gfCNCPoint2[28765] = {X 324.3107, Y 48.3200, Z -3.8333, A 0.000, B 0.000, C 0.000 }
gfCNCPoint2[28766] = {X 325.5555, Y 48.4004, Z -3.8333, A 0.000, B 0.000, C 0.000 }
gfCNCPoint2[28767] = {X 326.7797, Y 48.6402, Z -3.8333, A 0.000, B 0.000, C 0.000 }
gfCNCPoint2[28768] = {X 325.5882, Y 48.0963, Z -3.8333, A 0.000, B 0.000, C 0.000 }
gfCNCPoint2[28769] = {X 324.4810, Y 47.3966, Z -3.8333, A 0.000, B 0.000, C 0.000 }
gfCNCPoint2[28770] = {X 323.4784, Y 46.5538, Z -3.8333, A 0.000, B 0.000, C 0.000 }
gfCNCPoint2[28771] = {X 322.8382, Y 45.9295, Z -3.8333, A 0.000, B 0.000, C 0.000 }
gfCNCPoint2[28772] = {X 322.2180, Y 45.2650, Z -3.8333, A 0.000, B 0.000, C 0.000 }
gfCNCPoint2[28773] = {X 321.6628, Y 44.5452, Z -3.8333, A 0.000, B 0.000, C 0.000 }
gfCNCPoint2[28774] = {X 323.6300, Y 43.1703, Z -3.8333, A 0.000, B 0.000, C 0.000 }
gfCNCPoint2[28775] = {X 323.0063, Y 42.0918, Z -3.8333, A 0.000, B 0.000, C 0.000 }
gfCNCPoint2[28776] = {X 322.5757, Y 40.9227, Z -3.8333, A 0.000, B 0.000, C 0.000 }
gfCNCPoint2[28777] = {X 322.3506, Y 39.6973, Z -3.8333, A 0.000, B 0.000, C 0.000 }
gfCNCPoint2[28778] = {X 322.3379, Y 38.4514, Z -3.8333, A 0.000, B 0.000, C 0.000 }
gfCNCPoint2[28779] = {X 322.5377, Y 37.2217, Z -3.8333, A 0.000, B 0.000, C 0.000 }
gfCNCPoint2[28780] = {X 322.9443, Y 36.0440, Z -3.8333, A 0.000, B 0.000, C 0.000 }
gfCNCPoint2[28781] = {X 323.5458, Y 34.9529, Z -3.8333, A 0.000, B 0.000, C 0.000 }
gfCNCPoint2[28782] = {X 327.7841, Y 28.6157, Z -3.8333, A 0.000, B 0.000, C 0.000 }
gfCNCPoint2[28783] = {X 328.5200, Y 27.6906, Z -3.8333, A 0.000, B 0.000, C 0.000 }
gfCNCPoint2[28784] = {X 329.3960, Y 26.8968, Z -3.8333, A 0.000, B 0.000, C 0.000 }
gfCNCPoint2[28785] = {X 330.3889, Y 26.2552, Z -3.8333, A 0.000, B 0.000, C 0.000 }
gfCNCPoint2[28786] = {X 331.5063, Y 25.7713, Z -3.8333, A 0.000, B 0.000, C 0.000 }
gfCNCPoint2[28787] = {X 332.6887, Y 25.4804, Z -3.8333, A 0.000, B 0.000, C 0.000 }
gfCNCPoint2[28788] = {X 333.9031, Y 25.3907, Z -3.8333, A 0.000, B 0.000, C 0.000 }
gfCNCPoint2[28789] = {X 335.1154, Y 25.5046, Z -3.8333, A 0.000, B 0.000, C 0.000 }
gfCNCPoint2[28790] = {X 336.2918, Y 25.8191, Z -3.8333, A 0.000, B 0.000, C 0.000 }
gfCNCPoint2[28791] = {X 337.3993, Y 26.3252, Z -3.8333, A 0.000, B 0.000, C 0.000 }
gfCNCPoint2[28792] = {X 338.1754, Y 26.8291, Z -3.8333, A 0.000, B 0.000, C 0.000 }
gfCNCPoint2[28793] = {X 338.8813, Y 27.4275, Z -3.8333, A 0.000, B 0.000, C 0.000 }
gfCNCPoint2[28794] = {X 339.5028, Y 28.0267, Z -3.8333, A 0.000, B 0.000, C 0.000 }
gfCNCPoint2[28795] = {X 340.3314, Y 28.9977, Z -3.8333, A 0.000, B 0.000, C 0.000 }
gfCNCPoint2[28796] = {X 340.9777, Y 30.0985, Z -3.8333, A 0.000, B 0.000, C 0.000 }
gfCNCPoint2[28797] = {X 341.4218, Y 31.2952, Z -3.8333, A 0.000, B 0.000, C 0.000 }
gfCNCPoint2[28798] = {X 341.6500, Y 32.5511, Z -3.8333, A 0.000, B 0.000, C 0.000 }
gfCNCPoint2[28799] = {X 341.8446, Y 32.7091, Z -3.8333, A 0.000, B 0.000, C 0.000 }
gfCNCPoint2[28800] = {X 342.0414, Y 32.8643, Z -3.8333, A 0.000, B 0.000, C 0.000 }
gfCNCPoint2[28801] = {X 342.9843, Y 33.4816, Z -3.8333, A 0.000, B 0.000, C 0.000 }
gfCNCPoint2[28802] = {X 344.0076, Y 33.9537, Z -3.8333, A 0.000, B 0.000, C 0.000 }
gfCNCPoint2[28803] = {X 345.0891, Y 34.2705, Z -3.8333, A 0.000, B 0.000, C 0.000 }
gfCNCPoint2[28804] = {X 346.2053, Y 34.4251, Z -3.8333, A 0.000, B 0.000, C 0.000 }
gfCNCPoint2[28805] = {X 347.3322, Y 34.4141, Z -3.8333, A 0.000, B 0.000, C 0.000 }
gfCNCPoint2[28806] = {X 348.3018, Y 34.2887, Z -3.8333, A 0.000, B 0.000, C 0.000 }
gfCNCPoint2[28807] = {X 349.2376, Y 34.0059, Z -3.8333, A 0.000, B 0.000, C 0.000 }
gfCNCPoint2[28808] = {X 350.1143, Y 33.5732, Z -3.8333, A 0.000, B 0.000, C 0.000 }
gfCNCPoint2[28809] = {X 350.9081, Y 33.0025, Z -3.8333, A 0.000, B 0.000, C 0.000 }
gfCNCPoint2[28810] = {X 351.7847, Y 32.1513, Z -3.8333, A 0.000, B 0.000, C 0.000 }
gfCNCPoint2[28811] = {X 352.5434, Y 31.1936, Z -3.8333, A 0.000, B 0.000, C 0.000 }
gfCNCPoint2[28812] = {X 353.1716, Y 30.1456, Z -3.8333, A 0.000, B 0.000, C 0.000 }
gfCNCPoint2[28813] = {X 353.6586, Y 29.0250, Z -3.8333, A 0.000, B 0.000, C 0.000 }
gfCNCPoint2[28814] = {X 353.9962, Y 27.8507, Z -3.8333, A 0.000, B 0.000, C 0.000 }
gfCNCPoint2[28815] = {X 354.2236, Y 26.4407, Z -3.8333, A 0.000, B 0.000, C 0.000 }
gfCNCPoint2[28816] = {X 354.3157, Y 25.0155, Z -3.8333, A 0.000, B 0.000, C 0.000 }
gfCNCPoint2[28817] = {X 354.2717, Y 23.5880, Z -3.8333, A 0.000, B 0.000, C 0.000 }
gfCNCPoint2[28818] = {X 354.0919, Y 22.1712, Z -3.8333, A 0.000, B 0.000, C 0.000 }
gfCNCPoint2[28819] = {X 353.8393, Y 21.0759, Z -3.8333, A 0.000, B 0.000, C 0.000 }
gfCNCPoint2[28820] = {X 353.4527, Y 20.0204, Z -3.8333, A 0.000, B 0.000, C 0.000 }
gfCNCPoint2[28821] = {X 352.9380, Y 19.0210, Z -3.8333, A 0.000, B 0.000, C 0.000 }
gfCNCPoint2[28822] = {X 352.3033, Y 18.0933, Z -3.8333, A 0.000, B 0.000, C 0.000 }
gfCNCPoint2[28823] = {X 351.5364, Y 17.2660, Z -3.8333, A 0.000, B 0.000, C 0.000 }
gfCNCPoint2[28824] = {X 350.6339, Y 16.5894, Z -3.8333, A 0.000, B 0.000, C 0.000 }
gfCNCPoint2[28825] = {X 349.6248, Y 16.0851, Z -3.8333, A 0.000, B 0.000, C 0.000 }
gfCNCPoint2[28826] = {X 348.5418, Y 15.7695, Z -3.8333, A 0.000, B 0.000, C 0.000 }
gfCNCPoint2[28827] = {X 347.1561, Y 15.5988, Z -3.8333, A 0.000, B 0.000, C 0.000 }
gfCNCPoint2[28828] = {X 345.7600, Y 15.6149, Z -3.8333, A 0.000, B 0.000, C 0.000 }
gfCNCPoint2[28829] = {X 344.3786, Y 15.8174, Z -3.8333, A 0.000, B 0.000, C 0.000 }
gfCNCPoint2[28830] = {X 343.0366, Y 16.2027, Z -3.8333, A 0.000, B 0.000, C 0.000 }
gfCNCPoint2[28831] = {X 341.7582, Y 16.7639, Z -3.8333, A 0.000, B 0.000, C 0.000 }
gfCNCPoint2[28832] = {X 341.4305, Y 17.8589, Z -3.8333, A 0.000, B 0.000, C 0.000 }
gfCNCPoint2[28833] = {X 340.9355, Y 18.8891, Z -3.8333, A 0.000, B 0.000, C 0.000 }
gfCNCPoint2[28834] = {X 340.2853, Y 19.8292, Z -3.8333, A 0.000, B 0.000, C 0.000 }
gfCNCPoint2[28835] = {X 345.8671, Y 24.3770, Z -3.8333, A 0.000, B 0.000, C 0.000 }
gfCNCPoint2[28836] = {X 346.4659, Y 25.2133, Z -3.8333, A 0.000, B 0.000, C 0.000 }
gfCNCPoint2[28837] = {X 347.0039, Y 26.0900, Z -3.8333, A 0.000, B 0.000, C 0.000 }
gfCNCPoint2[28838] = {X 347.1178, Y 24.7341, Z -3.8333, A 0.000, B 0.000, C 0.000 }
gfCNCPoint2[28839] = {X 346.9938, Y 23.3790, Z -3.8333, A 0.000, B 0.000, C 0.000 }
gfCNCPoint2[28840] = {X 346.9498, Y 23.1696, Z -3.8333, A 0.000, B 0.000, C 0.000 }
gfCNCPoint2[28841] = {X 346.8818, Y 22.9666, Z -3.8333, A 0.000, B 0.000, C 0.000 }
gfCNCPoint2[28842] = {X 346.3957, Y 23.6871, Z -3.8333, A 0.000, B 0.000, C 0.000 }
gfCNCPoint2[28843] = {X 345.8671, Y 24.3770, Z -3.8333, A 0.000, B 0.000, C 0.000 }
gfCNCPoint2[28844] = {X 344.0065, Y 22.8611, Z -3.8333, A 0.000, B 0.000, C 0.000 }
gfCNCPoint2[28845] = {X 343.3271, Y 23.6263, Z -3.8333, A 0.000, B 0.000, C 0.000 }
gfCNCPoint2[28846] = {X 342.5854, Y 24.3313, Z -3.8333, A 0.000, B 0.000, C 0.000 }
gfCNCPoint2[28847] = {X 342.8589, Y 24.5949, Z -3.8333, A 0.000, B 0.000, C 0.000 }
gfCNCPoint2[28848] = {X 343.9809, Y 25.8612, Z -3.8333, A 0.000, B 0.000, C 0.000 }
gfCNCPoint2[28849] = {X 344.9149, Y 27.2717, Z -3.8333, A 0.000, B 0.000, C 0.000 }
gfCNCPoint2[28850] = {X 345.4668, Y 28.3751, Z -3.8333, A 0.000, B 0.000, C 0.000 }
gfCNCPoint2[28851] = {X 345.9032, Y 29.5290, Z -3.8333, A 0.000, B 0.000, C 0.000 }
gfCNCPoint2[28852] = {X 346.4601, Y 29.6317, Z -3.8333, A 0.000, B 0.000, C 0.000 }
gfCNCPoint2[28853] = {X 347.0263, Y 29.6224, Z -3.8333, A 0.000, B 0.000, C 0.000 }
gfCNCPoint2[28854] = {X 347.4358, Y 29.5572, Z -3.8333, A 0.000, B 0.000, C 0.000 }
gfCNCPoint2[28855] = {X 347.7945, Y 29.3494, Z -3.8333, A 0.000, B 0.000, C 0.000 }
gfCNCPoint2[28856] = {X 348.4750, Y 28.6296, Z -3.8333, A 0.000, B 0.000, C 0.000 }
gfCNCPoint2[28857] = {X 348.9857, Y 27.7810, Z -3.8333, A 0.000, B 0.000, C 0.000 }
gfCNCPoint2[28858] = {X 349.3032, Y 26.8428, Z -3.8333, A 0.000, B 0.000, C 0.000 }
gfCNCPoint2[28859] = {X 349.3374, Y 26.6713, Z -3.8333, A 0.000, B 0.000, C 0.000 }
gfCNCPoint2[28860] = {X 349.3687, Y 26.4992, Z -3.8333, A 0.000, B 0.000, C 0.000 }
gfCNCPoint2[28861] = {X 349.5021, Y 25.3279, Z -3.8333, A 0.000, B 0.000, C 0.000 }
gfCNCPoint2[28862] = {X 349.4993, Y 24.1490, Z -3.8333, A 0.000, B 0.000, C 0.000 }
gfCNCPoint2[28863] = {X 349.3602, Y 22.9783, Z -3.8333, A 0.000, B 0.000, C 0.000 }
gfCNCPoint2[28864] = {X 349.1884, Y 22.2867, Z -3.8333, A 0.000, B 0.000, C 0.000 }
gfCNCPoint2[28865] = {X 348.9031, Y 21.6337, Z -3.8333, A 0.000, B 0.000, C 0.000 }
gfCNCPoint2[28866] = {X 348.5124, Y 21.0377, Z -3.8333, A 0.000, B 0.000, C 0.000 }
gfCNCPoint2[28867] = {X 348.1200, Y 20.6785, Z -3.8333, A 0.000, B 0.000, C 0.000 }
gfCNCPoint2[28868] = {X 347.6259, Y 20.4813, Z -3.8333, A 0.000, B 0.000, C 0.000 }
gfCNCPoint2[28869] = {X 346.5728, Y 20.3828, Z -3.8333, A 0.000, B 0.000, C 0.000 }
gfCNCPoint2[28870] = {X 345.5198, Y 20.4831, Z -3.8333, A 0.000, B 0.000, C 0.000 }
gfCNCPoint2[28871] = {X 344.8328, Y 21.7164, Z -3.8333, A 0.000, B 0.000, C 0.000 }
gfCNCPoint2[28872] = {X 344.0065, Y 22.8611, Z -3.8333, A 0.000, B 0.000, C 0.000 }
gfCNCPoint2[28873] = {X 342.1459, Y 21.3451, Z -3.8333, A 0.000, B 0.000, C 0.000 }
gfCNCPoint2[28874] = {X 341.6015, Y 21.9583, Z -3.8333, A 0.000, B 0.000, C 0.000 }
gfCNCPoint2[28875] = {X 341.0072, Y 22.5232, Z -3.8333, A 0.000, B 0.000, C 0.000 }
gfCNCPoint2[28876] = {X 340.7216, Y 22.7630, Z -3.8333, A 0.000, B 0.000, C 0.000 }
gfCNCPoint2[28877] = {X 340.4270, Y 22.9916, Z -3.8333, A 0.000, B 0.000, C 0.000 }
gfCNCPoint2[28878] = {X 339.6615, Y 23.5549, Z -3.8333, A 0.000, B 0.000, C 0.000 }
gfCNCPoint2[28879] = {X 339.1299, Y 23.9121, Z -3.8333, A 0.000, B 0.000, C 0.000 }
gfCNCPoint2[28880] = {X 338.5759, Y 24.2333, Z -3.8333, A 0.000, B 0.000, C 0.000 }
gfCNCPoint2[28881] = {X 339.6078, Y 24.9035, Z -3.8333, A 0.000, B 0.000, C 0.000 }
gfCNCPoint2[28882] = {X 340.5464, Y 25.6991, Z -3.8333, A 0.000, B 0.000, C 0.000 }
gfCNCPoint2[28883] = {X 341.1848, Y 26.3148, Z -3.8333, A 0.000, B 0.000, C 0.000 }
gfCNCPoint2[28884] = {X 342.1201, Y 27.3790, Z -3.8333, A 0.000, B 0.000, C 0.000 }
gfCNCPoint2[28885] = {X 342.8900, Y 28.5683, Z -3.8333, A 0.000, B 0.000, C 0.000 }
gfCNCPoint2[28886] = {X 343.4780, Y 29.8572, Z -3.8333, A 0.000, B 0.000, C 0.000 }
gfCNCPoint2[28887] = {X 343.8716, Y 31.2182, Z -3.8333, A 0.000, B 0.000, C 0.000 }
gfCNCPoint2[28888] = {X 344.6368, Y 31.6212, Z -3.8333, A 0.000, B 0.000, C 0.000 }
gfCNCPoint2[28889] = {X 345.4577, Y 31.8932, Z -3.8333, A 0.000, B 0.000, C 0.000 }
gfCNCPoint2[28890] = {X 346.3121, Y 32.0269, Z -3.8333, A 0.000, B 0.000, C 0.000 }
gfCNCPoint2[28891] = {X 347.1768, Y 32.0187, Z -3.8333, A 0.000, B 0.000, C 0.000 }
gfCNCPoint2[28892] = {X 347.9590, Y 31.9040, Z -3.8333, A 0.000, B 0.000, C 0.000 }
gfCNCPoint2[28893] = {X 348.6962, Y 31.6182, Z -3.8333, A 0.000, B 0.000, C 0.000 }
gfCNCPoint2[28894] = {X 349.3514, Y 31.1758, Z -3.8333, A 0.000, B 0.000, C 0.000 }
gfCNCPoint2[28895] = {X 350.1528, Y 30.3722, Z -3.8333, A 0.000, B 0.000, C 0.000 }
gfCNCPoint2[28896] = {X 350.8138, Y 29.4496, Z -3.8333, A 0.000, B 0.000, C 0.000 }
gfCNCPoint2[28897] = {X 351.3172, Y 28.4324, Z -3.8333, A 0.000, B 0.000, C 0.000 }
gfCNCPoint2[28898] = {X 351.6496, Y 27.3472, Z -3.8333, A 0.000, B 0.000, C 0.000 }
gfCNCPoint2[28899] = {X 351.8779, Y 25.7641, Z -3.8333, A 0.000, B 0.000, C 0.000 }
gfCNCPoint2[28900] = {X 351.9036, Y 24.1648, Z -3.8333, A 0.000, B 0.000, C 0.000 }
gfCNCPoint2[28901] = {X 351.7261, Y 22.5752, Z -3.8333, A 0.000, B 0.000, C 0.000 }
gfCNCPoint2[28902] = {X 351.4573, Y 21.5045, Z -3.8333, A 0.000, B 0.000, C 0.000 }
gfCNCPoint2[28903] = {X 351.0147, Y 20.4931, Z -3.8333, A 0.000, B 0.000, C 0.000 }
gfCNCPoint2[28904] = {X 350.4107, Y 19.5691, Z -3.8333, A 0.000, B 0.000, C 0.000 }
gfCNCPoint2[28905] = {X 349.7597, Y 18.9043, Z -3.8333, A 0.000, B 0.000, C 0.000 }
gfCNCPoint2[28906] = {X 348.9692, Y 18.4138, Z -3.8333, A 0.000, B 0.000, C 0.000 }
gfCNCPoint2[28907] = {X 348.0845, Y 18.1256, Z -3.8333, A 0.000, B 0.000, C 0.000 }
gfCNCPoint2[28908] = {X 346.9930, Y 17.9935, Z -3.8333, A 0.000, B 0.000, C 0.000 }
gfCNCPoint2[28909] = {X 345.8937, Y 18.0119, Z -3.8333, A 0.000, B 0.000, C 0.000 }
gfCNCPoint2[28910] = {X 344.8073, Y 18.1805, Z -3.8333, A 0.000, B 0.000, C 0.000 }
gfCNCPoint2[28911] = {X 343.7541, Y 18.4960, Z -3.8333, A 0.000, B 0.000, C 0.000 }
gfCNCPoint2[28912] = {X 343.3269, Y 19.5045, Z -3.8333, A 0.000, B 0.000, C 0.000 }
gfCNCPoint2[28913] = {X 342.7886, Y 20.4583, Z -3.8333, A 0.000, B 0.000, C 0.000 }
gfCNCPoint2[28914] = {X 342.1459, Y 21.3451, Z -3.8333, A 0.000, B 0.000, C 0.000 }
gfCNCPoint2[28915] = {X 340.2853, Y 19.8292, Z -3.8333, A 0.000, B 0.000, C 0.000 }
gfCNCPoint2[28916] = {X 339.6794, Y 20.4860, Z -3.8333, A 0.000, B 0.000, C 0.000 }
gfCNCPoint2[28917] = {X 338.9976, Y 21.0636, Z -3.8333, A 0.000, B 0.000, C 0.000 }
gfCNCPoint2[28918] = {X 338.2497, Y 21.6140, Z -3.8333, A 0.000, B 0.000, C 0.000 }
gfCNCPoint2[28919] = {X 337.8538, Y 21.8795, Z -3.8333, A 0.000, B 0.000, C 0.000 }
gfCNCPoint2[28920] = {X 337.4413, Y 22.1185, Z -3.8333, A 0.000, B 0.000, C 0.000 }
gfCNCPoint2[28921] = {X 336.3239, Y 22.6023, Z -3.8333, A 0.000, B 0.000, C 0.000 }
gfCNCPoint2[28922] = {X 335.1415, Y 22.8932, Z -3.8333, A 0.000, B 0.000, C 0.000 }
gfCNCPoint2[28923] = {X 333.9271, Y 22.9829, Z -3.8333, A 0.000, B 0.000, C 0.000 }
gfCNCPoint2[28924] = {X 332.7148, Y 22.8690, Z -3.8333, A 0.000, B 0.000, C 0.000 }
gfCNCPoint2[28925] = {X 331.5384, Y 22.5546, Z -3.8333, A 0.000, B 0.000, C 0.000 }
gfCNCPoint2[28926] = {X 330.4309, Y 22.0485, Z -3.8333, A 0.000, B 0.000, C 0.000 }
gfCNCPoint2[28927] = {X 329.5143, Y 21.4374, Z -3.8333, A 0.000, B 0.000, C 0.000 }
gfCNCPoint2[28928] = {X 328.7005, Y 20.6949, Z -3.8333, A 0.000, B 0.000, C 0.000 }
gfCNCPoint2[28929] = {X 328.0080, Y 19.8382, Z -3.8333, A 0.000, B 0.000, C 0.000 }
gfCNCPoint2[28930] = {X 327.4528, Y 18.8869, Z -3.8333, A 0.000, B 0.000, C 0.000 }
gfCNCPoint2[28931] = {X 323.9321, Y 11.6443, Z -3.8333, A 0.000, B 0.000, C 0.000 }
gfCNCPoint2[28932] = {X 323.5337, Y 10.6422, Z -3.8333, A 0.000, B 0.000, C 0.000 }
gfCNCPoint2[28933] = {X 323.2878, Y 9.5922, Z -3.8333, A 0.000, B 0.000, C 0.000 }
gfCNCPoint2[28934] = {X 323.1997, Y 8.5174, Z -3.8333, A 0.000, B 0.000, C 0.000 }
gfCNCPoint2[28935] = {X 323.2713, Y 7.4413, Z -3.8333, A 0.000, B 0.000, C 0.000 }
gfCNCPoint2[28936] = {X 323.4720, Y 6.4885, Z -3.8333, A 0.000, B 0.000, C 0.000 }
gfCNCPoint2[28937] = {X 323.7980, Y 5.5709, Z -3.8333, A 0.000, B 0.000, C 0.000 }
gfCNCPoint2[28938] = {X 324.2435, Y 4.7050, Z -3.8333, A 0.000, B 0.000, C 0.000 }
gfCNCPoint2[28939] = {X 168.0205, Y 4.7050, Z -3.8333, A 0.000, B 0.000, C 0.000 }
gfCNCPoint2[28940] = {X 168.0205, Y 9.5050, Z -3.8333, A 0.000, B 0.000, C 0.000 }
gfCNCPoint2[28941] = {X 166.5360, Y 9.5050, Z -3.8333, A 0.000, B 0.000, C 0.000 }
gfCNCPoint2[28942] = {X 166.5855, Y 9.9931, Z -3.8333, A 0.000, B 0.000, C 0.000 }
gfCNCPoint2[28943] = {X 166.6021, Y 10.4835, Z -3.8333, A 0.000, B 0.000, C 0.000 }
gfCNCPoint2[28944] = {X 166.6021, Y 13.0969, Z -3.8333, A 0.000, B 0.000, C 0.000 }
gfCNCPoint2[28945] = {X 166.8569, Y 11.8210, Z -3.8333, A 0.000, B 0.000, C 0.000 }
gfCNCPoint2[28946] = {X 167.3348, Y 10.6108, Z -3.8333, A 0.000, B 0.000, C 0.000 }
gfCNCPoint2[28947] = {X 168.0205, Y 9.5050, Z -3.8333, A 0.000, B 0.000, C 0.000 }
gfCNCPoint2[28948] = {X 168.0205, Y 7.1050, Z -3.8333, A 0.000, B 0.000, C 0.000 }
gfCNCPoint2[28949] = {X 162.8435, Y 7.1050, Z -3.8333, A 0.000, B 0.000, C 0.000 }
gfCNCPoint2[28950] = {X 163.4703, Y 7.9131, Z -3.8333, A 0.000, B 0.000, C 0.000 }
gfCNCPoint2[28951] = {X 163.9149, Y 8.8341, Z -3.8333, A 0.000, B 0.000, C 0.000 }
gfCNCPoint2[28952] = {X 164.1578, Y 9.8276, Z -3.8333, A 0.000, B 0.000, C 0.000 }
gfCNCPoint2[28953] = {X 164.1910, Y 10.1548, Z -3.8333, A 0.000, B 0.000, C 0.000 }
gfCNCPoint2[28954] = {X 164.2021, Y 10.4835, Z -3.8333, A 0.000, B 0.000, C 0.000 }
gfCNCPoint2[28955] = {X 164.2021, Y 17.4615, Z -3.8333, A 0.000, B 0.000, C 0.000 }
gfCNCPoint2[28956] = {X 164.1139, Y 18.3848, Z -3.8333, A 0.000, B 0.000, C 0.000 }
gfCNCPoint2[28957] = {X 163.8527, Y 19.2747, Z -3.8333, A 0.000, B 0.000, C 0.000 }
gfCNCPoint2[28958] = {X 163.4279, Y 20.0992, Z -3.8333, A 0.000, B 0.000, C 0.000 }
gfCNCPoint2[28959] = {X 162.8547, Y 20.8283, Z -3.8333, A 0.000, B 0.000, C 0.000 }
gfCNCPoint2[28960] = {X 162.1539, Y 21.4359, Z -3.8333, A 0.000, B 0.000, C 0.000 }
gfCNCPoint2[28961] = {X 161.3508, Y 21.8998, Z -3.8333, A 0.000, B 0.000, C 0.000 }
gfCNCPoint2[28962] = {X 160.4745, Y 22.2035, Z -3.8333, A 0.000, B 0.000, C 0.000 }
gfCNCPoint2[28963] = {X 162.1747, Y 29.1999, Z -3.8333, A 0.000, B 0.000, C 0.000 }
gfCNCPoint2[28964] = {X 161.1123, Y 29.4081, Z -3.8333, A 0.000, B 0.000, C 0.000 }
gfCNCPoint2[28965] = {X 160.0356, Y 29.5204, Z -3.8333, A 0.000, B 0.000, C 0.000 }
gfCNCPoint2[28966] = {X 160.0350, Y 38.3365, Z -3.8333, A 0.000, B 0.000, C 0.000 }
gfCNCPoint2[28967] = {X 160.6830, Y 39.6933, Z -3.8333, A 0.000, B 0.000, C 0.000 }
gfCNCPoint2[28968] = {X 161.1580, Y 41.1200, Z -3.8333, A 0.000, B 0.000, C 0.000 }
gfCNCPoint2[28969] = {X 162.0480, Y 41.1200, Z -3.8333, A 0.000, B 0.000, C 0.000 }
gfCNCPoint2[28970] = {X 161.6737, Y 39.3706, Z -3.8333, A 0.000, B 0.000, C 0.000 }
gfCNCPoint2[28971] = {X 161.4498, Y 37.5957, Z -3.8333, A 0.000, B 0.000, C 0.000 }
gfCNCPoint2[28972] = {X 161.3316, Y 35.4804, Z -3.8333, A 0.000, B 0.000, C 0.000 }
gfCNCPoint2[28973] = {X 161.4138, Y 33.3634, Z -3.8333, A 0.000, B 0.000, C 0.000 }
gfCNCPoint2[28974] = {X 161.6957, Y 31.2636, Z -3.8333, A 0.000, B 0.000, C 0.000 }
gfCNCPoint2[28975] = {X 162.1747, Y 29.1999, Z -3.8333, A 0.000, B 0.000, C 0.000 }
gfCNCPoint2[28976] = {X 161.6080, Y 26.8678, Z -3.8333, A 0.000, B 0.000, C 0.000 }
gfCNCPoint2[28977] = {X 160.4732, Y 27.0728, Z -3.8333, A 0.000, B 0.000, C 0.000 }
gfCNCPoint2[28978] = {X 159.3221, Y 27.1415, Z -3.8333, A 0.000, B 0.000, C 0.000 }
gfCNCPoint2[28979] = {X 158.6554, Y 27.1415, Z -3.8333, A 0.000, B 0.000, C 0.000 }
gfCNCPoint2[28980] = {X 158.1448, Y 27.1258, Z -3.8333, A 0.000, B 0.000, C 0.000 }
gfCNCPoint2[28981] = {X 157.6357, Y 27.0833, Z -3.8333, A 0.000, B 0.000, C 0.000 }
gfCNCPoint2[28982] = {X 157.6349, Y 38.9960, Z -3.8333, A 0.000, B 0.000, C 0.000 }
gfCNCPoint2[28983] = {X 158.2188, Y 40.0484, Z -3.8333, A 0.000, B 0.000, C 0.000 }
gfCNCPoint2[28984] = {X 158.6680, Y 41.1649, Z -3.8333, A 0.000, B 0.000, C 0.000 }
gfCNCPoint2[28985] = {X 158.9759, Y 42.3283, Z -3.8333, A 0.000, B 0.000, C 0.000 }
gfCNCPoint2[28986] = {X 159.1375, Y 43.5209, Z -3.8333, A 0.000, B 0.000, C 0.000 }
gfCNCPoint2[28987] = {X 159.2980, Y 43.5200, Z -3.8333, A 0.000, B 0.000, C 0.000 }
gfCNCPoint2[28988] = {X 165.4299, Y 43.5200, Z -3.8333, A 0.000, B 0.000, C 0.000 }
gfCNCPoint2[28989] = {X 164.8363, Y 42.0419, Z -3.8333, A 0.000, B 0.000, C 0.000 }
gfCNCPoint2[28990] = {X 164.3714, Y 40.5184, Z -3.8333, A 0.000, B 0.000, C 0.000 }
gfCNCPoint2[28991] = {X 164.0379, Y 38.9571, Z -3.8333, A 0.000, B 0.000, C 0.000 }
gfCNCPoint2[28992] = {X 163.8396, Y 37.3729, Z -3.8333, A 0.000, B 0.000, C 0.000 }
gfCNCPoint2[28993] = {X 163.7317, Y 35.4783, Z -3.8333, A 0.000, B 0.000, C 0.000 }
gfCNCPoint2[28994] = {X 163.8039, Y 33.5820, Z -3.8333, A 0.000, B 0.000, C 0.000 }
gfCNCPoint2[28995] = {X 164.0555, Y 31.7011, Z -3.8333, A 0.000, B 0.000, C 0.000 }
gfCNCPoint2[28996] = {X 164.4843, Y 29.8525, Z -3.8333, A 0.000, B 0.000, C 0.000 }
gfCNCPoint2[28997] = {X 164.8363, Y 28.7332, Z -3.8333, A 0.000, B 0.000, C 0.000 }
gfCNCPoint2[28998] = {X 165.2534, Y 27.6365, Z -3.8333, A 0.000, B 0.000, C 0.000 }
gfCNCPoint2[28999] = {X 165.8700, Y 26.3057, Z -3.8333, A 0.000, B 0.000, C 0.000 }
gfCNCPoint2[29000] = {X 166.6043, Y 25.0361, Z -3.8333, A 0.000, B 0.000, C 0.000 }
gfCNCPoint2[29001] = {X 167.4503, Y 23.8379, Z -3.8333, A 0.000, B 0.000, C 0.000 }
gfCNCPoint2[29002] = {X 167.1640, Y 23.1367, Z -3.8333, A 0.000, B 0.000, C 0.000 }
gfCNCPoint2[29003] = {X 166.2873, Y 24.1837, Z -3.8333, A 0.000, B 0.000, C 0.000 }
gfCNCPoint2[29004] = {X 165.2721, Y 25.0970, Z -3.8333, A 0.000, B 0.000, C 0.000 }
gfCNCPoint2[29005] = {X 164.1384, Y 25.8583, Z -3.8333, A 0.000, B 0.000, C 0.000 }
gfCNCPoint2[29006] = {X 162.9089, Y 26.4525, Z -3.8333, A 0.000, B 0.000, C 0.000 }
gfCNCPoint2[29007] = {X 161.6080, Y 26.8678, Z -3.8333, A 0.000, B 0.000, C 0.000 }
gfCNCPoint2[29008] = {X 161.0412, Y 24.5356, Z -3.8333, A 0.000, B 0.000, C 0.000 }
gfCNCPoint2[29009] = {X 160.1878, Y 24.6899, Z -3.8333, A 0.000, B 0.000, C 0.000 }
gfCNCPoint2[29010] = {X 159.3221, Y 24.7415, Z -3.8333, A 0.000, B 0.000, C 0.000 }
gfCNCPoint2[29011] = {X 158.6660, Y 24.7415, Z -3.8333, A 0.000, B 0.000, C 0.000 }
gfCNCPoint2[29012] = {X 158.2815, Y 24.7297, Z -3.8333, A 0.000, B 0.000, C 0.000 }
gfCNCPoint2[29013] = {X 157.8982, Y 24.6977, Z -3.8333, A 0.000, B 0.000, C 0.000 }
gfCNCPoint2[29014] = {X 156.9779, Y 24.5364, Z -3.8333, A 0.000, B 0.000, C 0.000 }
gfCNCPoint2[29015] = {X 156.0856, Y 24.2591, Z -3.8333, A 0.000, B 0.000, C 0.000 }
gfCNCPoint2[29016] = {X 155.2360, Y 23.8704, Z -3.8333, A 0.000, B 0.000, C 0.000 }
gfCNCPoint2[29017] = {X 155.2349, Y 39.7518, Z -3.8333, A 0.000, B 0.000, C 0.000 }
gfCNCPoint2[29018] = {X 155.8256, Y 40.6437, Z -3.8333, A 0.000, B 0.000, C 0.000 }
gfCNCPoint2[29019] = {X 156.2800, Y 41.6123, Z -3.8333, A 0.000, B 0.000, C 0.000 }
gfCNCPoint2[29020] = {X 156.5883, Y 42.6368, Z -3.8333, A 0.000, B 0.000, C 0.000 }
gfCNCPoint2[29021] = {X 156.7438, Y 43.6953, Z -3.8333, A 0.000, B 0.000, C 0.000 }
gfCNCPoint2[29022] = {X 156.7578, Y 43.9475, Z -3.8333, A 0.000, B 0.000, C 0.000 }
gfCNCPoint2[29023] = {X 156.7631, Y 44.2001, Z -3.8333, A 0.000, B 0.000, C 0.000 }
gfCNCPoint2[29024] = {X 156.7629, Y 45.0587, Z -3.8333, A 0.000, B 0.000, C 0.000 }
gfCNCPoint2[29025] = {X 156.7352, Y 45.6370, Z -3.8333, A 0.000, B 0.000, C 0.000 }
gfCNCPoint2[29026] = {X 156.6616, Y 46.2112, Z -3.8333, A 0.000, B 0.000, C 0.000 }
gfCNCPoint2[29027] = {X 157.9053, Y 46.0006, Z -3.8333, A 0.000, B 0.000, C 0.000 }
gfCNCPoint2[29028] = {X 159.1641, Y 45.9207, Z -3.8333, A 0.000, B 0.000, C 0.000 }
gfCNCPoint2[29029] = {X 159.2310, Y 45.9202, Z -3.8333, A 0.000, B 0.000, C 0.000 }
gfCNCPoint2[29030] = {X 159.2980, Y 45.9200, Z -3.8333, A 0.000, B 0.000, C 0.000 }
gfCNCPoint2[29031] = {X 169.6833, Y 45.9200, Z -3.8333, A 0.000, B 0.000, C 0.000 }
gfCNCPoint2[29032] = {X 168.9026, Y 44.8481, Z -3.8333, A 0.000, B 0.000, C 0.000 }
gfCNCPoint2[29033] = {X 168.2121, Y 43.7159, Z -3.8333, A 0.000, B 0.000, C 0.000 }
gfCNCPoint2[29034] = {X 167.6167, Y 42.5310, Z -3.8333, A 0.000, B 0.000, C 0.000 }
gfCNCPoint2[29035] = {X 166.9487, Y 40.7946, Z -3.8333, A 0.000, B 0.000, C 0.000 }
gfCNCPoint2[29036] = {X 166.4842, Y 38.9930, Z -3.8333, A 0.000, B 0.000, C 0.000 }
gfCNCPoint2[29037] = {X 166.2294, Y 37.1501, Z -3.8333, A 0.000, B 0.000, C 0.000 }
gfCNCPoint2[29038] = {X 166.1311, Y 35.3976, Z -3.8333, A 0.000, B 0.000, C 0.000 }
gfCNCPoint2[29039] = {X 166.2079, Y 33.6441, Z -3.8333, A 0.000, B 0.000, C 0.000 }
gfCNCPoint2[29040] = {X 166.4591, Y 31.9069, Z -3.8333, A 0.000, B 0.000, C 0.000 }
gfCNCPoint2[29041] = {X 166.8820, Y 30.2034, Z -3.8333, A 0.000, B 0.000, C 0.000 }
gfCNCPoint2[29042] = {X 167.4726, Y 28.5505, Z -3.8333, A 0.000, B 0.000, C 0.000 }
gfCNCPoint2[29043] = {X 168.2334, Y 26.9813, Z -3.8333, A 0.000, B 0.000, C 0.000 }
gfCNCPoint2[29044] = {X 169.1857, Y 25.5205, Z -3.8333, A 0.000, B 0.000, C 0.000 }
gfCNCPoint2[29045] = {X 170.3144, Y 24.1911, Z -3.8333, A 0.000, B 0.000, C 0.000 }
gfCNCPoint2[29046] = {X 169.9865, Y 23.6224, Z -3.8333, A 0.000, B 0.000, C 0.000 }
gfCNCPoint2[29047] = {X 169.7113, Y 23.0264, Z -3.8333, A 0.000, B 0.000, C 0.000 }
gfCNCPoint2[29048] = {X 167.1001, Y 16.6309, Z -3.8333, A 0.000, B 0.000, C 0.000 }
gfCNCPoint2[29049] = {X 166.7820, Y 15.6636, Z -3.8333, A 0.000, B 0.000, C 0.000 }
gfCNCPoint2[29050] = {X 166.6021, Y 14.6613, Z -3.8333, A 0.000, B 0.000, C 0.000 }
gfCNCPoint2[29051] = {X 166.6021, Y 17.4615, Z -3.8333, A 0.000, B 0.000, C 0.000 }
gfCNCPoint2[29052] = {X 166.5130, Y 18.5970, Z -3.8333, A 0.000, B 0.000, C 0.000 }
gfCNCPoint2[29053] = {X 166.2479, Y 19.7047, Z -3.8333, A 0.000, B 0.000, C 0.000 }
gfCNCPoint2[29054] = {X 165.8132, Y 20.7575, Z -3.8333, A 0.000, B 0.000, C 0.000 }
gfCNCPoint2[29055] = {X 165.2197, Y 21.7296, Z -3.8333, A 0.000, B 0.000, C 0.000 }
gfCNCPoint2[29056] = {X 164.3787, Y 22.6988, Z -3.8333, A 0.000, B 0.000, C 0.000 }
gfCNCPoint2[29057] = {X 163.3807, Y 23.5052, Z -3.8333, A 0.000, B 0.000, C 0.000 }
gfCNCPoint2[29058] = {X 162.2565, Y 24.1239, Z -3.8333, A 0.000, B 0.000, C 0.000 }
gfCNCPoint2[29059] = {X 161.0412, Y 24.5356, Z -3.8333, A 0.000, B 0.000, C 0.000 }
gfCNCPoint2[29060] = {X 160.4745, Y 22.2035, Z -3.8333, A 0.000, B 0.000, C 0.000 }
gfCNCPoint2[29061] = {X 159.9024, Y 22.3069, Z -3.8333, A 0.000, B 0.000, C 0.000 }
gfCNCPoint2[29062] = {X 159.3221, Y 22.3415, Z -3.8333, A 0.000, B 0.000, C 0.000 }
gfCNCPoint2[29063] = {X 158.6766, Y 22.3415, Z -3.8333, A 0.000, B 0.000, C 0.000 }
gfCNCPoint2[29064] = {X 157.8799, Y 22.2730, Z -3.8333, A 0.000, B 0.000, C 0.000 }
gfCNCPoint2[29065] = {X 157.1047, Y 22.0761, Z -3.8333, A 0.000, B 0.000, C 0.000 }
gfCNCPoint2[29066] = {X 156.3718, Y 21.7562, Z -3.8333, A 0.000, B 0.000, C 0.000 }
gfCNCPoint2[29067] = {X 155.5229, Y 21.1783, Z -3.8333, A 0.000, B 0.000, C 0.000 }
gfCNCPoint2[29068] = {X 154.8126, Y 20.4367, Z -3.8333, A 0.000, B 0.000, C 0.000 }
gfCNCPoint2[29069] = {X 152.8362, Y 20.4376, Z -3.8333, A 0.000, B 0.000, C 0.000 }
gfCNCPoint2[29070] = {X 152.8348, Y 40.6542, Z -3.8333, A 0.000, B 0.000, C 0.000 }
gfCNCPoint2[29071] = {X 153.1753, Y 41.0225, Z -3.8333, A 0.000, B 0.000, C 0.000 }
gfCNCPoint2[29072] = {X 153.6797, Y 41.7264, Z -3.8333, A 0.000, B 0.000, C 0.000 }
gfCNCPoint2[29073] = {X 154.0528, Y 42.5079, Z -3.8333, A 0.000, B 0.000, C 0.000 }
gfCNCPoint2[29074] = {X 154.2830, Y 43.3428, Z -3.8333, A 0.000, B 0.000, C 0.000 }
gfCNCPoint2[29075] = {X 154.3631, Y 44.2051, Z -3.8333, A 0.000, B 0.000, C 0.000 }
gfCNCPoint2[29076] = {X 154.3629, Y 45.0469, Z -3.8333, A 0.000, B 0.000, C 0.000 }
gfCNCPoint2[29077] = {X 154.3441, Y 45.4307, Z -3.8333, A 0.000, B 0.000, C 0.000 }
gfCNCPoint2[29078] = {X 154.2951, Y 45.8119, Z -3.8333, A 0.000, B 0.000, C 0.000 }
gfCNCPoint2[29079] = {X 154.0370, Y 46.7541, Z -3.8333, A 0.000, B 0.000, C 0.000 }
gfCNCPoint2[29080] = {X 153.5963, Y 47.6260, Z -3.8333, A 0.000, B 0.000, C 0.000 }
gfCNCPoint2[29081] = {X 152.9909, Y 48.3926, Z -3.8333, A 0.000, B 0.000, C 0.000 }
gfCNCPoint2[29082] = {X 152.2448, Y 49.0233, Z -3.8333, A 0.000, B 0.000, C 0.000 }
gfCNCPoint2[29083] = {X 151.3881, Y 49.4928, Z -3.8333, A 0.000, B 0.000, C 0.000 }
gfCNCPoint2[29084] = {X 150.4551, Y 49.7822, Z -3.8333, A 0.000, B 0.000, C 0.000 }
gfCNCPoint2[29085] = {X 149.4831, Y 49.8800, Z -3.8333, A 0.000, B 0.000, C 0.000 }
gfCNCPoint2[29086] = {X 143.0396, Y 49.8800, Z -3.8333, A 0.000, B 0.000, C 0.000 }
gfCNCPoint2[29087] = {X 142.0923, Y 49.7872, Z -3.8333, A 0.000, B 0.000, C 0.000 }
gfCNCPoint2[29088] = {X 141.1811, Y 49.5122, Z -3.8333, A 0.000, B 0.000, C 0.000 }
gfCNCPoint2[29089] = {X 140.3405, Y 49.0656, Z -3.8333, A 0.000, B 0.000, C 0.000 }
gfCNCPoint2[29090] = {X 139.6026, Y 48.4643, Z -3.8333, A 0.000, B 0.000, C 0.000 }
gfCNCPoint2[29091] = {X 138.9955, Y 47.7312, Z -3.8333, A 0.000, B 0.000, C 0.000 }
gfCNCPoint2[29092] = {X 138.5423, Y 46.8942, Z -3.8333, A 0.000, B 0.000, C 0.000 }
gfCNCPoint2[29093] = {X 138.2601, Y 45.9852, Z -3.8333, A 0.000, B 0.000, C 0.000 }
gfCNCPoint2[29094] = {X 138.1598, Y 45.0386, Z -3.8333, A 0.000, B 0.000, C 0.000 }
gfCNCPoint2[29095] = {X 138.1601, Y 44.1416, Z -3.8333, A 0.000, B 0.000, C 0.000 }
gfCNCPoint2[29096] = {X 138.2148, Y 43.4769, Z -3.8333, A 0.000, B 0.000, C 0.000 }
gfCNCPoint2[29097] = {X 138.3597, Y 42.8258, Z -3.8333, A 0.000, B 0.000, C 0.000 }
gfCNCPoint2[29098] = {X 129.1532, Y 40.1052, Z -3.8333, A 0.000, B 0.000, C 0.000 }
gfCNCPoint2[29099] = {X 129.5665, Y 38.9035, Z -3.8333, A 0.000, B 0.000, C 0.000 }
gfCNCPoint2[29100] = {X 130.0836, Y 37.7426, Z -3.8333, A 0.000, B 0.000, C 0.000 }
gfCNCPoint2[29101] = {X 130.0836, Y 31.6021, Z -3.8333, A 0.000, B 0.000, C 0.000 }
gfCNCPoint2[29102] = {X 129.2061, Y 31.3797, Z -3.8333, A 0.000, B 0.000, C 0.000 }
gfCNCPoint2[29103] = {X 128.3442, Y 31.1029, Z -3.8333, A 0.000, B 0.000, C 0.000 }
gfCNCPoint2[29104] = {X 128.3439, Y 38.3287, Z -3.8333, A 0.000, B 0.000, C 0.000 }
gfCNCPoint2[29105] = {X 128.7845, Y 39.2006, Z -3.8333, A 0.000, B 0.000, C 0.000 }
gfCNCPoint2[29106] = {X 129.1532, Y 40.1052, Z -3.8333, A 0.000, B 0.000, C 0.000 }
gfCNCPoint2[29107] = {X 131.4548, Y 40.7854, Z -3.8333, A 0.000, B 0.000, C 0.000 }
gfCNCPoint2[29108] = {X 131.9017, Y 39.5320, Z -3.8333, A 0.000, B 0.000, C 0.000 }
gfCNCPoint2[29109] = {X 132.4836, Y 38.3354, Z -3.8333, A 0.000, B 0.000, C 0.000 }
gfCNCPoint2[29110] = {X 132.4836, Y 29.5202, Z -3.8333, A 0.000, B 0.000, C 0.000 }
gfCNCPoint2[29111] = {X 131.3524, Y 29.3993, Z -3.8333, A 0.000, B 0.000, C 0.000 }
gfCNCPoint2[29112] = {X 130.2377, Y 29.1725, Z -3.8333, A 0.000, B 0.000, C 0.000 }
gfCNCPoint2[29113] = {X 129.1492, Y 28.8419, Z -3.8333, A 0.000, B 0.000, C 0.000 }
gfCNCPoint2[29114] = {X 128.0248, Y 28.3765, Z -3.8333, A 0.000, B 0.000, C 0.000 }
gfCNCPoint2[29115] = {X 126.9529, Y 27.8004, Z -3.8333, A 0.000, B 0.000, C 0.000 }
gfCNCPoint2[29116] = {X 125.9444, Y 27.1194, Z -3.8333, A 0.000, B 0.000, C 0.000 }
gfCNCPoint2[29117] = {X 125.9438, Y 38.9893, Z -3.8333, A 0.000, B 0.000, C 0.000 }
gfCNCPoint2[29118] = {X 126.4738, Y 39.9284, Z -3.8333, A 0.000, B 0.000, C 0.000 }
gfCNCPoint2[29119] = {X 126.8960, Y 40.9205, Z -3.8333, A 0.000, B 0.000, C 0.000 }
gfCNCPoint2[29120] = {X 127.2098, Y 41.9730, Z -3.8333, A 0.000, B 0.000, C 0.000 }
gfCNCPoint2[29121] = {X 127.4025, Y 43.0542, Z -3.8333, A 0.000, B 0.000, C 0.000 }
gfCNCPoint2[29122] = {X 127.4714, Y 44.1502, Z -3.8333, A 0.000, B 0.000, C 0.000 }
gfCNCPoint2[29123] = {X 127.4716, Y 45.0000, Z -3.8333, A 0.000, B 0.000, C 0.000 }
gfCNCPoint2[29124] = {X 127.4070, Y 46.1159, Z -3.8333, A 0.000, B 0.000, C 0.000 }
gfCNCPoint2[29125] = {X 127.2143, Y 47.2168, Z -3.8333, A 0.000, B 0.000, C 0.000 }
gfCNCPoint2[29126] = {X 126.8960, Y 48.2883, Z -3.8333, A 0.000, B 0.000, C 0.000 }
gfCNCPoint2[29127] = {X 126.2883, Y 49.6376, Z -3.8333, A 0.000, B 0.000, C 0.000 }
gfCNCPoint2[29128] = {X 125.4821, Y 50.8786, Z -3.8333, A 0.000, B 0.000, C 0.000 }
gfCNCPoint2[29129] = {X 124.4962, Y 51.9821, Z -3.8333, A 0.000, B 0.000, C 0.000 }
gfCNCPoint2[29130] = {X 123.3536, Y 52.9225, Z -3.8333, A 0.000, B 0.000, C 0.000 }
gfCNCPoint2[29131] = {X 122.0810, Y 53.6778, Z -3.8333, A 0.000, B 0.000, C 0.000 }
gfCNCPoint2[29132] = {X 120.7081, Y 54.2302, Z -3.8333, A 0.000, B 0.000, C 0.000 }
gfCNCPoint2[29133] = {X 119.2671, Y 54.5669, Z -3.8333, A 0.000, B 0.000, C 0.000 }
gfCNCPoint2[29134] = {X 117.7916, Y 54.6800, Z -3.8333, A 0.000, B 0.000, C 0.000 }
gfCNCPoint2[29135] = {X 111.9185, Y 54.6800, Z -3.8333, A 0.000, B 0.000, C 0.000 }
gfCNCPoint2[29136] = {X 110.6386, Y 54.5950, Z -3.8333, A 0.000, B 0.000, C 0.000 }
gfCNCPoint2[29137] = {X 109.3812, Y 54.3415, Z -3.8333, A 0.000, B 0.000, C 0.000 }
gfCNCPoint2[29138] = {X 108.1683, Y 53.9240, Z -3.8333, A 0.000, B 0.000, C 0.000 }
gfCNCPoint2[29139] = {X 107.0213, Y 53.3498, Z -3.8333, A 0.000, B 0.000, C 0.000 }
gfCNCPoint2[29140] = {X 106.6480, Y 53.5578, Z -3.8333, A 0.000, B 0.000, C 0.000 }
gfCNCPoint2[29141] = {X 106.2658, Y 53.7492, Z -3.8333, A 0.000, B 0.000, C 0.000 }
gfCNCPoint2[29142] = {X 105.0149, Y 54.2383, Z -3.8333, A 0.000, B 0.000, C 0.000 }
gfCNCPoint2[29143] = {X 103.7084, Y 54.5495, Z -3.8333, A 0.000, B 0.000, C 0.000 }
gfCNCPoint2[29144] = {X 102.3713, Y 54.6768, Z -3.8333, A 0.000, B 0.000, C 0.000 }
gfCNCPoint2[29145] = {X 101.0295, Y 54.6179, Z -3.8333, A 0.000, B 0.000, C 0.000 }
gfCNCPoint2[29146] = {X 99.7088, Y 54.3738, Z -3.8333, A 0.000, B 0.000, C 0.000 }
gfCNCPoint2[29147] = {X 98.4345, Y 53.9493, Z -3.8333, A 0.000, B 0.000, C 0.000 }
gfCNCPoint2[29148] = {X 97.2313, Y 53.3524, Z -3.8333, A 0.000, B 0.000, C 0.000 }
gfCNCPoint2[29149] = {X 96.0852, Y 53.9255, Z -3.8333, A 0.000, B 0.000, C 0.000 }
gfCNCPoint2[29150] = {X 94.8734, Y 54.3422, Z -3.8333, A 0.000, B 0.000, C 0.000 }
gfCNCPoint2[29151] = {X 93.6172, Y 54.5952, Z -3.8333, A 0.000, B 0.000, C 0.000 }
gfCNCPoint2[29152] = {X 92.3385, Y 54.6800, Z -3.8333, A 0.000, B 0.000, C 0.000 }
gfCNCPoint2[29153] = {X 85.8951, Y 54.6800, Z -3.8333, A 0.000, B 0.000, C 0.000 }
gfCNCPoint2[29154] = {X 84.6159, Y 54.5951, Z -3.8333, A 0.000, B 0.000, C 0.000 }
gfCNCPoint2[29155] = {X 83.3592, Y 54.3419, Z -3.8333, A 0.000, B 0.000, C 0.000 }
gfCNCPoint2[29156] = {X 82.1469, Y 53.9249, Z -3.8333, A 0.000, B 0.000, C 0.000 }
gfCNCPoint2[29157] = {X 81.0644, Y 55.1572, Z -3.8333, A 0.000, B 0.000, C 0.000 }
gfCNCPoint2[29158] = {X 79.8495, Y 56.2591, Z -3.8333, A 0.000, B 0.000, C 0.000 }
gfCNCPoint2[29159] = {X 78.5178, Y 57.2166, Z -3.8333, A 0.000, B 0.000, C 0.000 }
gfCNCPoint2[29160] = {X 77.0863, Y 58.0174, Z -3.8333, A 0.000, B 0.000, C 0.000 }
gfCNCPoint2[29161] = {X 75.5734, Y 58.6511, Z -3.8333, A 0.000, B 0.000, C 0.000 }
gfCNCPoint2[29162] = {X 73.9986, Y 59.1096, Z -3.8333, A 0.000, B 0.000, C 0.000 }
gfCNCPoint2[29163] = {X 72.3820, Y 59.3871, Z -3.8333, A 0.000, B 0.000, C 0.000 }
gfCNCPoint2[29164] = {X 70.7445, Y 59.4800, Z -3.8333, A 0.000, B 0.000, C 0.000 }
gfCNCPoint2[29165] = {X 64.1851, Y 59.4800, Z -3.8333, A 0.000, B 0.000, C 0.000 }
gfCNCPoint2[29166] = {X 62.4203, Y 59.3720, Z -3.8333, A 0.000, B 0.000, C 0.000 }
gfCNCPoint2[29167] = {X 60.6818, Y 59.0498, Z -3.8333, A 0.000, B 0.000, C 0.000 }
gfCNCPoint2[29168] = {X 58.9955, Y 58.5181, Z -3.8333, A 0.000, B 0.000, C 0.000 }
gfCNCPoint2[29169] = {X 57.3866, Y 57.7848, Z -3.8333, A 0.000, B 0.000, C 0.000 }
gfCNCPoint2[29170] = {X 55.8790, Y 56.8608, Z -3.8333, A 0.000, B 0.000, C 0.000 }
gfCNCPoint2[29171] = {X 54.3715, Y 57.7848, Z -3.8333, A 0.000, B 0.000, C 0.000 }
gfCNCPoint2[29172] = {X 52.7626, Y 58.5181, Z -3.8333, A 0.000, B 0.000, C 0.000 }
gfCNCPoint2[29173] = {X 51.0763, Y 59.0498, Z -3.8333, A 0.000, B 0.000, C 0.000 }
gfCNCPoint2[29174] = {X 49.3378, Y 59.3720, Z -3.8333, A 0.000, B 0.000, C 0.000 }
gfCNCPoint2[29175] = {X 47.5729, Y 59.4800, Z -3.8333, A 0.000, B 0.000, C 0.000 }
gfCNCPoint2[29176] = {X 40.6393, Y 59.4800, Z -3.8333, A 0.000, B 0.000, C 0.000 }
gfCNCPoint2[29177] = {X 38.9796, Y 59.3846, Z -3.8333, A 0.000, B 0.000, C 0.000 }
gfCNCPoint2[29178] = {X 37.3418, Y 59.0995, Z -3.8333, A 0.000, B 0.000, C 0.000 }
gfCNCPoint2[29179] = {X 35.7474, Y 58.6286, Z -3.8333, A 0.000, B 0.000, C 0.000 }
gfCNCPoint2[29180] = {X 34.0329, Y 59.4869, Z -3.8333, A 0.000, B 0.000, C 0.000 }
gfCNCPoint2[29181] = {X 32.2400, Y 60.1662, Z -3.8333, A 0.000, B 0.000, C 0.000 }
gfCNCPoint2[29182] = {X 30.3872, Y 60.6596, Z -3.8333, A 0.000, B 0.000, C 0.000 }
gfCNCPoint2[29183] = {X 28.4938, Y 60.9618, Z -3.8333, A 0.000, B 0.000, C 0.000 }
gfCNCPoint2[29184] = {X 26.3374, Y 61.8556, Z -3.8333, A 0.000, B 0.000, C 0.000 }
gfCNCPoint2[29185] = {X 24.1361, Y 62.6325, Z -3.8333, A 0.000, B 0.000, C 0.000 }
gfCNCPoint2[29186] = {X 21.7294, Y 63.3344, Z -3.8333, A 0.000, B 0.000, C 0.000 }
gfCNCPoint2[29187] = {X 19.2810, Y 63.8733, Z -3.8333, A 0.000, B 0.000, C 0.000 }
gfCNCPoint2[29188] = {X 16.8020, Y 64.2465, Z -3.8333, A 0.000, B 0.000, C 0.000 }
gfCNCPoint2[29189] = {X 14.3035, Y 64.4526, Z -3.8333, A 0.000, B 0.000, C 0.000 }
gfCNCPoint2[29190] = {X 14.3035, Y 85.6950, Z -3.8333, A 0.000, B 0.000, C 0.000 }
gfCNCPoint2[29191] = {X 112.5232, Y 85.6950, Z -3.8333, A 0.000, B 0.000, C 0.000 }
gfCNCPoint2[29192] = {X 113.6258, Y 84.5917, Z -3.8333, A 0.000, B 0.000, C 0.000 }
gfCNCPoint2[29193] = {X 114.8256, Y 83.5948, Z -3.8333, A 0.000, B 0.000, C 0.000 }
gfCNCPoint2[29194] = {X 116.1122, Y 82.7130, Z -3.8333, A 0.000, B 0.000, C 0.000 }
gfCNCPoint2[29195] = {X 117.4748, Y 81.9537, Z -3.8333, A 0.000, B 0.000, C 0.000 }
gfCNCPoint2[29196] = {X 111.0539, Y 69.0645, Z -3.8333, A 0.000, B 0.000, C 0.000 }
gfCNCPoint2[29197] = {X 109.0273, Y 68.9058, Z -3.8333, A 0.000, B 0.000, C 0.000 }
gfCNCPoint2[29198] = {X 107.0213, Y 68.5768, Z -3.8333, A 0.000, B 0.000, C 0.000 }
gfCNCPoint2[29199] = {X 105.0765, Y 68.8983, Z -3.8333, A 0.000, B 0.000, C 0.000 }
gfCNCPoint2[29200] = {X 103.1119, Y 69.0597, Z -3.8333, A 0.000, B 0.000, C 0.000 }
gfCNCPoint2[29201] = {X 101.1407, Y 69.0599, Z -3.8333, A 0.000, B 0.000, C 0.000 }
gfCNCPoint2[29202] = {X 99.1761, Y 68.8989, Z -3.8333, A 0.000, B 0.000, C 0.000 }
gfCNCPoint2[29203] = {X 97.2313, Y 68.5777, Z -3.8333, A 0.000, B 0.000, C 0.000 }
gfCNCPoint2[29204] = {X 95.6131, Y 68.8563, Z -3.8333, A 0.000, B 0.000, C 0.000 }
gfCNCPoint2[29205] = {X 93.9796, Y 69.0240, Z -3.8333, A 0.000, B 0.000, C 0.000 }
gfCNCPoint2[29206] = {X 92.3385, Y 69.0800, Z -3.8333, A 0.000, B 0.000, C 0.000 }
gfCNCPoint2[29207] = {X 86.6884, Y 69.0800, Z -3.8333, A 0.000, B 0.000, C 0.000 }
gfCNCPoint2[29208] = {X 84.7317, Y 70.2668, Z -3.8333, A 0.000, B 0.000, C 0.000 }
gfCNCPoint2[29209] = {X 82.6871, Y 71.2950, Z -3.8333, A 0.000, B 0.000, C 0.000 }
gfCNCPoint2[29210] = {X 107.2684, Y 71.2950, Z -3.8333, A 0.000, B 0.000, C 0.000 }
gfCNCPoint2[29211] = {X 109.1219, Y 70.1132, Z -3.8333, A 0.000, B 0.000, C 0.000 }
gfCNCPoint2[29212] = {X 111.0539, Y 69.0645, Z -3.8333, A 0.000, B 0.000, C 0.000 }
gfCNCPoint2[29213] = {X 112.1240, Y 71.2127, Z -3.8333, A 0.000, B 0.000, C 0.000 }
gfCNCPoint2[29214] = {X 113.1266, Y 70.7371, Z -3.8333, A 0.000, B 0.000, C 0.000 }
gfCNCPoint2[29215] = {X 114.1466, Y 70.3003, Z -3.8333, A 0.000, B 0.000, C 0.000 }
gfCNCPoint2[29216] = {X 117.4434, Y 66.6800, Z -3.8333, A 0.000, B 0.000, C 0.000 }
gfCNCPoint2[29217] = {X 111.9185, Y 66.6800, Z -3.8333, A 0.000, B 0.000, C 0.000 }
gfCNCPoint2[29218] = {X 111.5292, Y 66.6765, Z -3.8333, A 0.000, B 0.000, C 0.000 }
gfCNCPoint2[29219] = {X 111.1400, Y 66.6660, Z -3.8333, A 0.000, B 0.000, C 0.000 }
gfCNCPoint2[29220] = {X 109.0675, Y 66.4917, Z -3.8333, A 0.000, B 0.000, C 0.000 }
gfCNCPoint2[29221] = {X 107.0213, Y 66.1197, Z -3.8333, A 0.000, B 0.000, C 0.000 }
gfCNCPoint2[29222] = {X 105.0796, Y 66.4776, Z -3.8333, A 0.000, B 0.000, C 0.000 }
gfCNCPoint2[29223] = {X 103.1135, Y 66.6574, Z -3.8333, A 0.000, B 0.000, C 0.000 }
gfCNCPoint2[29224] = {X 101.1392, Y 66.6576, Z -3.8333, A 0.000, B 0.000, C 0.000 }
gfCNCPoint2[29225] = {X 99.1730, Y 66.4782, Z -3.8333, A 0.000, B 0.000, C 0.000 }
gfCNCPoint2[29226] = {X 97.2313, Y 66.1207, Z -3.8333, A 0.000, B 0.000, C 0.000 }
gfCNCPoint2[29227] = {X 95.6161, Y 66.4308, Z -3.8333, A 0.000, B 0.000, C 0.000 }
gfCNCPoint2[29228] = {X 93.9821, Y 66.6176, Z -3.8333, A 0.000, B 0.000, C 0.000 }
gfCNCPoint2[29229] = {X 92.3385, Y 66.6800, Z -3.8333, A 0.000, B 0.000, C 0.000 }
gfCNCPoint2[29230] = {X 85.9487, Y 66.6800, Z -3.8333, A 0.000, B 0.000, C 0.000 }
gfCNCPoint2[29231] = {X 83.8780, Y 67.9935, Z -3.8333, A 0.000, B 0.000, C 0.000 }
gfCNCPoint2[29232] = {X 81.6947, Y 69.1098, Z -3.8333, A 0.000, B 0.000, C 0.000 }
gfCNCPoint2[29233] = {X 79.6017, Y 69.9548, Z -3.8333, A 0.000, B 0.000, C 0.000 }
gfCNCPoint2[29234] = {X 77.4443, Y 70.6184, Z -3.8333, A 0.000, B 0.000, C 0.000 }
gfCNCPoint2[29235] = {X 75.2382, Y 71.0959, Z -3.8333, A 0.000, B 0.000, C 0.000 }
gfCNCPoint2[29236] = {X 72.9995, Y 71.3838, Z -3.8333, A 0.000, B 0.000, C 0.000 }
gfCNCPoint2[29237] = {X 70.7445, Y 71.4800, Z -3.8333, A 0.000, B 0.000, C 0.000 }
gfCNCPoint2[29238] = {X 64.1851, Y 71.4800, Z -3.8333, A 0.000, B 0.000, C 0.000 }
gfCNCPoint2[29239] = {X 62.0752, Y 71.3958, Z -3.8333, A 0.000, B 0.000, C 0.000 }
gfCNCPoint2[29240] = {X 59.9787, Y 71.1438, Z -3.8333, A 0.000, B 0.000, C 0.000 }
gfCNCPoint2[29241] = {X 57.9089, Y 70.7255, Z -3.8333, A 0.000, B 0.000, C 0.000 }
gfCNCPoint2[29242] = {X 55.8790, Y 70.1436, Z -3.8333, A 0.000, B 0.000, C 0.000 }
gfCNCPoint2[29243] = {X 53.8492, Y 70.7255, Z -3.8333, A 0.000, B 0.000, C 0.000 }
gfCNCPoint2[29244] = {X 51.7794, Y 71.1438, Z -3.8333, A 0.000, B 0.000, C 0.000 }
gfCNCPoint2[29245] = {X 49.6829, Y 71.3958, Z -3.8333, A 0.000, B 0.000, C 0.000 }
gfCNCPoint2[29246] = {X 47.5729, Y 71.4800, Z -3.8333, A 0.000, B 0.000, C 0.000 }
gfCNCPoint2[29247] = {X 40.6393, Y 71.4800, Z -3.8333, A 0.000, B 0.000, C 0.000 }
gfCNCPoint2[29248] = {X 38.8048, Y 71.4164, Z -3.8333, A 0.000, B 0.000, C 0.000 }
gfCNCPoint2[29249] = {X 36.9790, Y 71.2258, Z -3.8333, A 0.000, B 0.000, C 0.000 }
gfCNCPoint2[29250] = {X 34.4002, Y 72.0344, Z -3.8333, A 0.000, B 0.000, C 0.000 }
gfCNCPoint2[29251] = {X 31.7605, Y 72.6140, Z -3.8333, A 0.000, B 0.000, C 0.000 }
gfCNCPoint2[29252] = {X 30.3334, Y 73.1743, Z -3.8333, A 0.000, B 0.000, C 0.000 }
gfCNCPoint2[29253] = {X 28.8913, Y 73.6950, Z -3.8333, A 0.000, B 0.000, C 0.000 }
gfCNCPoint2[29254] = {X 108.0308, Y 73.6950, Z -3.8333, A 0.000, B 0.000, C 0.000 }
gfCNCPoint2[29255] = {X 110.0259, Y 72.3689, Z -3.8333, A 0.000, B 0.000, C 0.000 }
gfCNCPoint2[29256] = {X 112.1240, Y 71.2127, Z -3.8333, A 0.000, B 0.000, C 0.000 }
gfCNCPoint2[29257] = {X 113.1942, Y 73.3609, Z -3.8333, A 0.000, B 0.000, C 0.000 }
gfCNCPoint2[29258] = {X 114.3574, Y 72.8162, Z -3.8333, A 0.000, B 0.000, C 0.000 }
gfCNCPoint2[29259] = {X 115.5456, Y 72.3286, Z -3.8333, A 0.000, B 0.000, C 0.000 }
gfCNCPoint2[29260] = {X 123.7278, Y 63.3434, Z -3.8333, A 0.000, B 0.000, C 0.000 }
gfCNCPoint2[29261] = {X 121.7853, Y 63.8618, Z -3.8333, A 0.000, B 0.000, C 0.000 }
gfCNCPoint2[29262] = {X 119.7994, Y 64.1752, Z -3.8333, A 0.000, B 0.000, C 0.000 }
gfCNCPoint2[29263] = {X 117.7916, Y 64.2800, Z -3.8333, A 0.000, B 0.000, C 0.000 }
gfCNCPoint2[29264] = {X 111.9185, Y 64.2800, Z -3.8333, A 0.000, B 0.000, C 0.000 }
gfCNCPoint2[29265] = {X 110.2700, Y 64.2094, Z -3.8333, A 0.000, B 0.000, C 0.000 }
gfCNCPoint2[29266] = {X 108.6336, Y 63.9981, Z -3.8333, A 0.000, B 0.000, C 0.000 }
gfCNCPoint2[29267] = {X 107.0213, Y 63.6477, Z -3.8333, A 0.000, B 0.000, C 0.000 }
gfCNCPoint2[29268] = {X 105.0841, Y 64.0514, Z -3.8333, A 0.000, B 0.000, C 0.000 }
gfCNCPoint2[29269] = {X 103.1158, Y 64.2545, Z -3.8333, A 0.000, B 0.000, C 0.000 }
gfCNCPoint2[29270] = {X 101.1370, Y 64.2547, Z -3.8333, A 0.000, B 0.000, C 0.000 }
gfCNCPoint2[29271] = {X 99.1686, Y 64.0521, Z -3.8333, A 0.000, B 0.000, C 0.000 }
gfCNCPoint2[29272] = {X 97.2313, Y 63.6488, Z -3.8333, A 0.000, B 0.000, C 0.000 }
gfCNCPoint2[29273] = {X 95.6204, Y 63.9986, Z -3.8333, A 0.000, B 0.000, C 0.000 }
gfCNCPoint2[29274] = {X 93.9855, Y 64.2095, Z -3.8333, A 0.000, B 0.000, C 0.000 }
gfCNCPoint2[29275] = {X 92.3385, Y 64.2800, Z -3.8333, A 0.000, B 0.000, C 0.000 }
gfCNCPoint2[29276] = {X 85.8951, Y 64.2800, Z -3.8333, A 0.000, B 0.000, C 0.000 }
gfCNCPoint2[29277] = {X 85.5417, Y 64.2768, Z -3.8333, A 0.000, B 0.000, C 0.000 }
gfCNCPoint2[29278] = {X 85.1884, Y 64.2670, Z -3.8333, A 0.000, B 0.000, C 0.000 }
gfCNCPoint2[29279] = {X 83.3593, Y 65.5113, Z -3.8333, A 0.000, B 0.000, C 0.000 }
gfCNCPoint2[29280] = {X 81.4238, Y 66.5824, Z -3.8333, A 0.000, B 0.000, C 0.000 }
gfCNCPoint2[29281] = {X 79.3981, Y 67.4713, Z -3.8333, A 0.000, B 0.000, C 0.000 }
gfCNCPoint2[29282] = {X 77.2994, Y 68.1706, Z -3.8333, A 0.000, B 0.000, C 0.000 }
gfCNCPoint2[29283] = {X 75.1454, Y 68.6744, Z -3.8333, A 0.000, B 0.000, C 0.000 }
gfCNCPoint2[29284] = {X 72.9543, Y 68.9784, Z -3.8333, A 0.000, B 0.000, C 0.000 }
gfCNCPoint2[29285] = {X 70.7445, Y 69.0800, Z -3.8333, A 0.000, B 0.000, C 0.000 }
gfCNCPoint2[29286] = {X 64.1851, Y 69.0800, Z -3.8333, A 0.000, B 0.000, C 0.000 }
gfCNCPoint2[29287] = {X 62.0678, Y 68.9867, Z -3.8333, A 0.000, B 0.000, C 0.000 }
gfCNCPoint2[29288] = {X 59.9669, Y 68.7076, Z -3.8333, A 0.000, B 0.000, C 0.000 }
gfCNCPoint2[29289] = {X 57.8986, Y 68.2449, Z -3.8333, A 0.000, B 0.000, C 0.000 }
gfCNCPoint2[29290] = {X 55.8790, Y 67.6021, Z -3.8333, A 0.000, B 0.000, C 0.000 }
gfCNCPoint2[29291] = {X 53.8595, Y 68.2449, Z -3.8333, A 0.000, B 0.000, C 0.000 }
gfCNCPoint2[29292] = {X 51.7912, Y 68.7076, Z -3.8333, A 0.000, B 0.000, C 0.000 }
gfCNCPoint2[29293] = {X 49.6903, Y 68.9867, Z -3.8333, A 0.000, B 0.000, C 0.000 }
gfCNCPoint2[29294] = {X 47.5729, Y 69.0800, Z -3.8333, A 0.000, B 0.000, C 0.000 }
gfCNCPoint2[29295] = {X 40.6393, Y 69.0800, Z -3.8333, A 0.000, B 0.000, C 0.000 }
gfCNCPoint2[29296] = {X 38.6743, Y 68.9997, Z -3.8333, A 0.000, B 0.000, C 0.000 }
gfCNCPoint2[29297] = {X 36.7225, Y 68.7593, Z -3.8333, A 0.000, B 0.000, C 0.000 }
gfCNCPoint2[29298] = {X 34.8832, Y 69.3986, Z -3.8333, A 0.000, B 0.000, C 0.000 }
gfCNCPoint2[29299] = {X 33.0045, Y 69.9105, Z -3.8333, A 0.000, B 0.000, C 0.000 }
gfCNCPoint2[29300] = {X 31.0952, Y 70.2925, Z -3.8333, A 0.000, B 0.000, C 0.000 }
gfCNCPoint2[29301] = {X 29.6099, Y 70.8820, Z -3.8333, A 0.000, B 0.000, C 0.000 }
gfCNCPoint2[29302] = {X 28.1075, Y 71.4266, Z -3.8333, A 0.000, B 0.000, C 0.000 }
gfCNCPoint2[29303] = {X 27.6092, Y 71.5960, Z -3.8333, A 0.000, B 0.000, C 0.000 }
gfCNCPoint2[29304] = {X 27.1093, Y 71.7605, Z -3.8333, A 0.000, B 0.000, C 0.000 }
gfCNCPoint2[29305] = {X 25.5146, Y 72.2522, Z -3.8333, A 0.000, B 0.000, C 0.000 }
gfCNCPoint2[29306] = {X 23.9035, Y 72.6869, Z -3.8333, A 0.000, B 0.000, C 0.000 }
gfCNCPoint2[29307] = {X 23.9035, Y 76.0950, Z -3.8333, A 0.000, B 0.000, C 0.000 }
gfCNCPoint2[29308] = {X 108.8292, Y 76.0950, Z -3.8333, A 0.000, B 0.000, C 0.000 }
gfCNCPoint2[29309] = {X 110.2239, Y 75.0897, Z -3.8333, A 0.000, B 0.000, C 0.000 }
gfCNCPoint2[29310] = {X 111.6810, Y 74.1771, Z -3.8333, A 0.000, B 0.000, C 0.000 }
gfCNCPoint2[29311] = {X 113.1942, Y 73.3609, Z -3.8333, A 0.000, B 0.000, C 0.000 }
gfCNCPoint2[29312] = {X 114.2643, Y 75.5091, Z -3.8333, A 0.000, B 0.000, C 0.000 }
gfCNCPoint2[29313] = {X 115.5782, Y 74.9031, Z -3.8333, A 0.000, B 0.000, C 0.000 }
gfCNCPoint2[29314] = {X 116.9261, Y 74.3772, Z -3.8333, A 0.000, B 0.000, C 0.000 }
gfCNCPoint2[29315] = {X 130.4113, Y 59.5686, Z -3.8333, A 0.000, B 0.000, C 0.000 }
gfCNCPoint2[29316] = {X 129.5279, Y 58.7532, Z -3.8333, A 0.000, B 0.000, C 0.000 }
gfCNCPoint2[29317] = {X 128.6970, Y 57.8844, Z -3.8333, A 0.000, B 0.000, C 0.000 }
gfCNCPoint2[29318] = {X 127.3929, Y 58.8834, Z -3.8333, A 0.000, B 0.000, C 0.000 }
gfCNCPoint2[29319] = {X 125.9980, Y 59.7509, Z -3.8333, A 0.000, B 0.000, C 0.000 }
gfCNCPoint2[29320] = {X 124.5253, Y 60.4787, Z -3.8333, A 0.000, B 0.000, C 0.000 }
gfCNCPoint2[29321] = {X 122.9889, Y 61.0600, Z -3.8333, A 0.000, B 0.000, C 0.000 }
gfCNCPoint2[29322] = {X 121.2882, Y 61.5139, Z -3.8333, A 0.000, B 0.000, C 0.000 }
gfCNCPoint2[29323] = {X 119.5494, Y 61.7882, Z -3.8333, A 0.000, B 0.000, C 0.000 }
gfCNCPoint2[29324] = {X 117.7916, Y 61.8800, Z -3.8333, A 0.000, B 0.000, C 0.000 }
gfCNCPoint2[29325] = {X 111.9185, Y 61.8800, Z -3.8333, A 0.000, B 0.000, C 0.000 }
gfCNCPoint2[29326] = {X 110.2649, Y 61.7988, Z -3.8333, A 0.000, B 0.000, C 0.000 }
gfCNCPoint2[29327] = {X 108.6273, Y 61.5560, Z -3.8333, A 0.000, B 0.000, C 0.000 }
gfCNCPoint2[29328] = {X 107.0213, Y 61.1540, Z -3.8333, A 0.000, B 0.000, C 0.000 }
gfCNCPoint2[29329] = {X 105.0907, Y 61.6173, Z -3.8333, A 0.000, B 0.000, C 0.000 }
gfCNCPoint2[29330] = {X 103.1191, Y 61.8506, Z -3.8333, A 0.000, B 0.000, C 0.000 }
gfCNCPoint2[29331] = {X 101.1337, Y 61.8509, Z -3.8333, A 0.000, B 0.000, C 0.000 }
gfCNCPoint2[29332] = {X 99.1620, Y 61.6181, Z -3.8333, A 0.000, B 0.000, C 0.000 }
gfCNCPoint2[29333] = {X 97.2313, Y 61.1553, Z -3.8333, A 0.000, B 0.000, C 0.000 }
gfCNCPoint2[29334] = {X 95.6267, Y 61.5566, Z -3.8333, A 0.000, B 0.000, C 0.000 }
gfCNCPoint2[29335] = {X 93.9906, Y 61.7990, Z -3.8333, A 0.000, B 0.000, C 0.000 }
gfCNCPoint2[29336] = {X 92.3385, Y 61.8800, Z -3.8333, A 0.000, B 0.000, C 0.000 }
gfCNCPoint2[29337] = {X 85.8951, Y 61.8800, Z -3.8333, A 0.000, B 0.000, C 0.000 }
gfCNCPoint2[29338] = {X 85.1609, Y 61.8640, Z -3.8333, A 0.000, B 0.000, C 0.000 }
gfCNCPoint2[29339] = {X 84.4280, Y 61.8161, Z -3.8333, A 0.000, B 0.000, C 0.000 }
gfCNCPoint2[29340] = {X 82.7247, Y 63.0692, Z -3.8333, A 0.000, B 0.000, C 0.000 }
gfCNCPoint2[29341] = {X 80.9073, Y 64.1504, Z -3.8333, A 0.000, B 0.000, C 0.000 }
gfCNCPoint2[29342] = {X 78.9932, Y 65.0494, Z -3.8333, A 0.000, B 0.000, C 0.000 }
gfCNCPoint2[29343] = {X 77.0007, Y 65.7577, Z -3.8333, A 0.000, B 0.000, C 0.000 }
gfCNCPoint2[29344] = {X 74.9487, Y 66.2685, Z -3.8333, A 0.000, B 0.000, C 0.000 }
gfCNCPoint2[29345] = {X 72.8566, Y 66.5769, Z -3.8333, A 0.000, B 0.000, C 0.000 }
gfCNCPoint2[29346] = {X 70.7445, Y 66.6800, Z -3.8333, A 0.000, B 0.000, C 0.000 }
gfCNCPoint2[29347] = {X 64.1851, Y 66.6800, Z -3.8333, A 0.000, B 0.000, C 0.000 }
gfCNCPoint2[29348] = {X 62.0576, Y 66.5754, Z -3.8333, A 0.000, B 0.000, C 0.000 }
gfCNCPoint2[29349] = {X 59.9505, Y 66.2624, Z -3.8333, A 0.000, B 0.000, C 0.000 }
gfCNCPoint2[29350] = {X 57.8844, Y 65.7442, Z -3.8333, A 0.000, B 0.000, C 0.000 }
gfCNCPoint2[29351] = {X 55.8790, Y 65.0258, Z -3.8333, A 0.000, B 0.000, C 0.000 }
gfCNCPoint2[29352] = {X 53.8737, Y 65.7442, Z -3.8333, A 0.000, B 0.000, C 0.000 }
gfCNCPoint2[29353] = {X 51.8075, Y 66.2624, Z -3.8333, A 0.000, B 0.000, C 0.000 }
gfCNCPoint2[29354] = {X 49.7005, Y 66.5754, Z -3.8333, A 0.000, B 0.000, C 0.000 }
gfCNCPoint2[29355] = {X 47.5729, Y 66.6800, Z -3.8333, A 0.000, B 0.000, C 0.000 }
gfCNCPoint2[29356] = {X 40.6393, Y 66.6800, Z -3.8333, A 0.000, B 0.000, C 0.000 }
gfCNCPoint2[29357] = {X 38.5445, Y 66.5786, Z -3.8333, A 0.000, B 0.000, C 0.000 }
gfCNCPoint2[29358] = {X 36.4693, Y 66.2752, Z -3.8333, A 0.000, B 0.000, C 0.000 }
gfCNCPoint2[29359] = {X 34.5054, Y 67.0008, Z -3.8333, A 0.000, B 0.000, C 0.000 }
gfCNCPoint2[29360] = {X 32.4894, Y 67.5661, Z -3.8333, A 0.000, B 0.000, C 0.000 }
gfCNCPoint2[29361] = {X 30.4346, Y 67.9675, Z -3.8333, A 0.000, B 0.000, C 0.000 }
gfCNCPoint2[29362] = {X 28.4165, Y 68.7665, Z -3.8333, A 0.000, B 0.000, C 0.000 }
gfCNCPoint2[29363] = {X 26.3660, Y 69.4785, Z -3.8333, A 0.000, B 0.000, C 0.000 }
gfCNCPoint2[29364] = {X 23.9531, Y 70.1951, Z -3.8333, A 0.000, B 0.000, C 0.000 }
gfCNCPoint2[29365] = {X 21.5035, Y 70.7743, Z -3.8333, A 0.000, B 0.000, C 0.000 }
gfCNCPoint2[29366] = {X 21.5035, Y 78.4950, Z -3.8333, A 0.000, B 0.000, C 0.000 }
gfCNCPoint2[29367] = {X 109.6690, Y 78.4950, Z -3.8333, A 0.000, B 0.000, C 0.000 }
gfCNCPoint2[29368] = {X 111.1236, Y 77.3841, Z -3.8333, A 0.000, B 0.000, C 0.000 }
gfCNCPoint2[29369] = {X 112.6583, Y 76.3869, Z -3.8333, A 0.000, B 0.000, C 0.000 }
gfCNCPoint2[29370] = {X 114.2643, Y 75.5091, Z -3.8333, A 0.000, B 0.000, C 0.000 }
gfCNCPoint2[29371] = {X 115.3345, Y 77.6573, Z -3.8333, A 0.000, B 0.000, C 0.000 }
gfCNCPoint2[29372] = {X 116.7876, Y 76.9990, Z -3.8333, A 0.000, B 0.000, C 0.000 }
gfCNCPoint2[29373] = {X 118.2852, Y 76.4493, Z -3.8333, A 0.000, B 0.000, C 0.000 }
gfCNCPoint2[29374] = {X 133.9635, Y 59.2323, Z -3.8333, A 0.000, B 0.000, C 0.000 }
gfCNCPoint2[29375] = {X 132.7156, Y 58.3548, Z -3.8333, A 0.000, B 0.000, C 0.000 }
gfCNCPoint2[29376] = {X 131.5521, Y 57.3681, Z -3.8333, A 0.000, B 0.000, C 0.000 }
gfCNCPoint2[29377] = {X 130.4824, Y 56.2805, Z -3.8333, A 0.000, B 0.000, C 0.000 }
gfCNCPoint2[29378] = {X 129.6655, Y 55.2988, Z -3.8333, A 0.000, B 0.000, C 0.000 }
gfCNCPoint2[29379] = {X 128.9251, Y 54.2582, Z -3.8333, A 0.000, B 0.000, C 0.000 }
gfCNCPoint2[29380] = {X 128.0750, Y 55.1942, Z -3.8333, A 0.000, B 0.000, C 0.000 }
gfCNCPoint2[29381] = {X 127.1464, Y 56.0525, Z -3.8333, A 0.000, B 0.000, C 0.000 }
gfCNCPoint2[29382] = {X 125.7915, Y 57.0695, Z -3.8333, A 0.000, B 0.000, C 0.000 }
gfCNCPoint2[29383] = {X 124.3270, Y 57.9212, Z -3.8333, A 0.000, B 0.000, C 0.000 }
gfCNCPoint2[29384] = {X 122.7731, Y 58.5961, Z -3.8333, A 0.000, B 0.000, C 0.000 }
gfCNCPoint2[29385] = {X 121.1510, Y 59.0849, Z -3.8333, A 0.000, B 0.000, C 0.000 }
gfCNCPoint2[29386] = {X 119.4828, Y 59.3809, Z -3.8333, A 0.000, B 0.000, C 0.000 }
gfCNCPoint2[29387] = {X 117.7916, Y 59.4800, Z -3.8333, A 0.000, B 0.000, C 0.000 }
gfCNCPoint2[29388] = {X 111.9185, Y 59.4800, Z -3.8333, A 0.000, B 0.000, C 0.000 }
gfCNCPoint2[29389] = {X 110.2569, Y 59.3844, Z -3.8333, A 0.000, B 0.000, C 0.000 }
gfCNCPoint2[29390] = {X 108.6173, Y 59.0987, Z -3.8333, A 0.000, B 0.000, C 0.000 }
gfCNCPoint2[29391] = {X 107.0213, Y 58.6267, Z -3.8333, A 0.000, B 0.000, C 0.000 }
gfCNCPoint2[29392] = {X 105.4260, Y 59.0985, Z -3.8333, A 0.000, B 0.000, C 0.000 }
gfCNCPoint2[29393] = {X 103.7872, Y 59.3842, Z -3.8333, A 0.000, B 0.000, C 0.000 }
gfCNCPoint2[29394] = {X 102.1264, Y 59.4800, Z -3.8333, A 0.000, B 0.000, C 0.000 }
gfCNCPoint2[29395] = {X 100.4656, Y 59.3847, Z -3.8333, A 0.000, B 0.000, C 0.000 }
gfCNCPoint2[29396] = {X 98.8267, Y 59.0996, Z -3.8333, A 0.000, B 0.000, C 0.000 }
gfCNCPoint2[29397] = {X 97.2313, Y 58.6283, Z -3.8333, A 0.000, B 0.000, C 0.000 }
gfCNCPoint2[29398] = {X 95.6367, Y 59.0994, Z -3.8333, A 0.000, B 0.000, C 0.000 }
gfCNCPoint2[29399] = {X 93.9986, Y 59.3845, Z -3.8333, A 0.000, B 0.000, C 0.000 }
gfCNCPoint2[29400] = {X 92.3385, Y 59.4800, Z -3.8333, A 0.000, B 0.000, C 0.000 }
gfCNCPoint2[29401] = {X 85.8951, Y 59.4800, Z -3.8333, A 0.000, B 0.000, C 0.000 }
gfCNCPoint2[29402] = {X 84.7780, Y 59.4368, Z -3.8333, A 0.000, B 0.000, C 0.000 }
gfCNCPoint2[29403] = {X 83.6677, Y 59.3077, Z -3.8333, A 0.000, B 0.000, C 0.000 }
gfCNCPoint2[29404] = {X 82.0978, Y 60.5827, Z -3.8333, A 0.000, B 0.000, C 0.000 }
gfCNCPoint2[29405] = {X 80.4031, Y 61.6862, Z -3.8333, A 0.000, B 0.000, C 0.000 }
gfCNCPoint2[29406] = {X 78.6021, Y 62.6061, Z -3.8333, A 0.000, B 0.000, C 0.000 }
gfCNCPoint2[29407] = {X 76.7146, Y 63.3324, Z -3.8333, A 0.000, B 0.000, C 0.000 }
gfCNCPoint2[29408] = {X 74.7614, Y 63.8569, Z -3.8333, A 0.000, B 0.000, C 0.000 }
gfCNCPoint2[29409] = {X 72.7640, Y 64.1739, Z -3.8333, A 0.000, B 0.000, C 0.000 }
gfCNCPoint2[29410] = {X 70.7445, Y 64.2800, Z -3.8333, A 0.000, B 0.000, C 0.000 }
gfCNCPoint2[29411] = {X 64.1851, Y 64.2800, Z -3.8333, A 0.000, B 0.000, C 0.000 }
gfCNCPoint2[29412] = {X 62.0428, Y 64.1606, Z -3.8333, A 0.000, B 0.000, C 0.000 }
gfCNCPoint2[29413] = {X 59.9269, Y 63.8039, Z -3.8333, A 0.000, B 0.000, C 0.000 }
gfCNCPoint2[29414] = {X 57.8638, Y 63.2143, Z -3.8333, A 0.000, B 0.000, C 0.000 }
gfCNCPoint2[29415] = {X 55.8790, Y 62.3991, Z -3.8333, A 0.000, B 0.000, C 0.000 }
gfCNCPoint2[29416] = {X 53.8942, Y 63.2143, Z -3.8333, A 0.000, B 0.000, C 0.000 }
gfCNCPoint2[29417] = {X 51.8311, Y 63.8039, Z -3.8333, A 0.000, B 0.000, C 0.000 }
gfCNCPoint2[29418] = {X 49.7153, Y 64.1606, Z -3.8333, A 0.000, B 0.000, C 0.000 }
gfCNCPoint2[29419] = {X 47.5729, Y 64.2800, Z -3.8333, A 0.000, B 0.000, C 0.000 }
gfCNCPoint2[29420] = {X 40.6393, Y 64.2800, Z -3.8333, A 0.000, B 0.000, C 0.000 }
gfCNCPoint2[29421] = {X 39.1547, Y 64.2228, Z -3.8333, A 0.000, B 0.000, C 0.000 }
gfCNCPoint2[29422] = {X 37.6790, Y 64.0514, Z -3.8333, A 0.000, B 0.000, C 0.000 }
gfCNCPoint2[29423] = {X 36.2208, Y 63.7669, Z -3.8333, A 0.000, B 0.000, C 0.000 }
gfCNCPoint2[29424] = {X 34.1364, Y 64.5939, Z -3.8333, A 0.000, B 0.000, C 0.000 }
gfCNCPoint2[29425] = {X 31.9829, Y 65.2196, Z -3.8333, A 0.000, B 0.000, C 0.000 }
gfCNCPoint2[29426] = {X 29.7798, Y 65.6381, Z -3.8333, A 0.000, B 0.000, C 0.000 }
gfCNCPoint2[29427] = {X 27.7192, Y 66.4651, Z -3.8333, A 0.000, B 0.000, C 0.000 }
gfCNCPoint2[29428] = {X 25.6227, Y 67.1965, Z -3.8333, A 0.000, B 0.000, C 0.000 }
gfCNCPoint2[29429] = {X 23.4786, Y 67.8375, Z -3.8333, A 0.000, B 0.000, C 0.000 }
gfCNCPoint2[29430] = {X 21.3035, Y 68.3639, Z -3.8333, A 0.000, B 0.000, C 0.000 }
gfCNCPoint2[29431] = {X 19.1035, Y 68.7739, Z -3.8333, A 0.000, B 0.000, C 0.000 }
gfCNCPoint2[29432] = {X 19.1035, Y 80.8950, Z -3.8333, A 0.000, B 0.000, C 0.000 }
gfCNCPoint2[29433] = {X 110.5576, Y 80.8950, Z -3.8333, A 0.000, B 0.000, C 0.000 }
gfCNCPoint2[29434] = {X 112.0516, Y 79.6753, Z -3.8333, A 0.000, B 0.000, C 0.000 }
gfCNCPoint2[29435] = {X 113.6481, Y 78.5932, Z -3.8333, A 0.000, B 0.000, C 0.000 }
gfCNCPoint2[29436] = {X 115.3345, Y 77.6573, Z -3.8333, A 0.000, B 0.000, C 0.000 }
gfCNCPoint2[29437] = {X 116.4046, Y 79.8055, Z -3.8333, A 0.000, B 0.000, C 0.000 }
gfCNCPoint2[29438] = {X 117.9836, Y 79.1054, Z -3.8333, A 0.000, B 0.000, C 0.000 }
gfCNCPoint2[29439] = {X 119.6188, Y 78.5493, Z -3.8333, A 0.000, B 0.000, C 0.000 }
gfCNCPoint2[29440] = {X 137.8573, Y 58.5209, Z -3.8333, A 0.000, B 0.000, C 0.000 }
gfCNCPoint2[29441] = {X 136.5225, Y 57.9305, Z -3.8333, A 0.000, B 0.000, C 0.000 }
gfCNCPoint2[29442] = {X 135.2539, Y 57.2087, Z -3.8333, A 0.000, B 0.000, C 0.000 }
gfCNCPoint2[29443] = {X 134.0100, Y 56.3197, Z -3.8333, A 0.000, B 0.000, C 0.000 }
gfCNCPoint2[29444] = {X 132.8667, Y 55.3045, Z -3.8333, A 0.000, B 0.000, C 0.000 }
gfCNCPoint2[29445] = {X 131.8368, Y 54.1743, Z -3.8333, A 0.000, B 0.000, C 0.000 }
gfCNCPoint2[29446] = {X 130.9319, Y 52.9419, Z -3.8333, A 0.000, B 0.000, C 0.000 }
gfCNCPoint2[29447] = {X 130.2147, Y 51.7225, Z -3.8333, A 0.000, B 0.000, C 0.000 }
gfCNCPoint2[29448] = {X 129.6199, Y 50.4390, Z -3.8333, A 0.000, B 0.000, C 0.000 }
gfCNCPoint2[29449] = {X 129.1532, Y 49.1035, Z -3.8333, A 0.000, B 0.000, C 0.000 }
gfCNCPoint2[29450] = {X 128.6036, Y 50.3877, Z -3.8333, A 0.000, B 0.000, C 0.000 }
gfCNCPoint2[29451] = {X 127.9093, Y 51.5998, Z -3.8333, A 0.000, B 0.000, C 0.000 }
gfCNCPoint2[29452] = {X 127.0798, Y 52.7237, Z -3.8333, A 0.000, B 0.000, C 0.000 }
gfCNCPoint2[29453] = {X 126.0417, Y 53.8239, Z -3.8333, A 0.000, B 0.000, C 0.000 }
gfCNCPoint2[29454] = {X 124.8743, Y 54.7858, Z -3.8333, A 0.000, B 0.000, C 0.000 }
gfCNCPoint2[29455] = {X 123.5958, Y 55.5942, Z -3.8333, A 0.000, B 0.000, C 0.000 }
gfCNCPoint2[29456] = {X 122.2263, Y 56.2365, Z -3.8333, A 0.000, B 0.000, C 0.000 }
gfCNCPoint2[29457] = {X 120.7872, Y 56.7027, Z -3.8333, A 0.000, B 0.000, C 0.000 }
gfCNCPoint2[29458] = {X 119.3012, Y 56.9853, Z -3.8333, A 0.000, B 0.000, C 0.000 }
gfCNCPoint2[29459] = {X 117.7916, Y 57.0800, Z -3.8333, A 0.000, B 0.000, C 0.000 }
gfCNCPoint2[29460] = {X 111.9185, Y 57.0800, Z -3.8333, A 0.000, B 0.000, C 0.000 }
gfCNCPoint2[29461] = {X 110.2431, Y 56.9633, Z -3.8333, A 0.000, B 0.000, C 0.000 }
gfCNCPoint2[29462] = {X 108.6001, Y 56.6153, Z -3.8333, A 0.000, B 0.000, C 0.000 }
gfCNCPoint2[29463] = {X 107.0213, Y 56.0428, Z -3.8333, A 0.000, B 0.000, C 0.000 }
gfCNCPoint2[29464] = {X 105.4432, Y 56.6151, Z -3.8333, A 0.000, B 0.000, C 0.000 }
gfCNCPoint2[29465] = {X 103.8010, Y 56.9630, Z -3.8333, A 0.000, B 0.000, C 0.000 }
gfCNCPoint2[29466] = {X 102.1265, Y 57.0800, Z -3.8333, A 0.000, B 0.000, C 0.000 }
gfCNCPoint2[29467] = {X 100.4519, Y 56.9637, Z -3.8333, A 0.000, B 0.000, C 0.000 }
gfCNCPoint2[29468] = {X 98.8096, Y 56.6164, Z -3.8333, A 0.000, B 0.000, C 0.000 }
gfCNCPoint2[29469] = {X 97.2313, Y 56.0448, Z -3.8333, A 0.000, B 0.000, C 0.000 }
gfCNCPoint2[29470] = {X 95.6538, Y 56.6162, Z -3.8333, A 0.000, B 0.000, C 0.000 }
gfCNCPoint2[29471] = {X 94.0123, Y 56.9635, Z -3.8333, A 0.000, B 0.000, C 0.000 }
gfCNCPoint2[29472] = {X 92.3385, Y 57.0800, Z -3.8333, A 0.000, B 0.000, C 0.000 }
gfCNCPoint2[29473] = {X 85.8951, Y 57.0800, Z -3.8333, A 0.000, B 0.000, C 0.000 }
gfCNCPoint2[29474] = {X 84.3894, Y 56.9858, Z -3.8333, A 0.000, B 0.000, C 0.000 }
gfCNCPoint2[29475] = {X 82.9073, Y 56.7047, Z -3.8333, A 0.000, B 0.000, C 0.000 }
gfCNCPoint2[29476] = {X 81.4846, Y 58.0224, Z -3.8333, A 0.000, B 0.000, C 0.000 }
gfCNCPoint2[29477] = {X 79.9203, Y 59.1682, Z -3.8333, A 0.000, B 0.000, C 0.000 }
gfCNCPoint2[29478] = {X 78.2348, Y 60.1271, Z -3.8333, A 0.000, B 0.000, C 0.000 }
gfCNCPoint2[29479] = {X 76.4504, Y 60.8864, Z -3.8333, A 0.000, B 0.000, C 0.000 }
gfCNCPoint2[29480] = {X 74.5908, Y 61.4359, Z -3.8333, A 0.000, B 0.000, C 0.000 }
gfCNCPoint2[29481] = {X 72.6804, Y 61.7686, Z -3.8333, A 0.000, B 0.000, C 0.000 }
gfCNCPoint2[29482] = {X 70.7445, Y 61.8800, Z -3.8333, A 0.000, B 0.000, C 0.000 }
gfCNCPoint2[29483] = {X 64.1851, Y 61.8800, Z -3.8333, A 0.000, B 0.000, C 0.000 }
gfCNCPoint2[29484] = {X 62.4514, Y 61.7907, Z -3.8333, A 0.000, B 0.000, C 0.000 }
gfCNCPoint2[29485] = {X 60.7359, Y 61.5238, Z -3.8333, A 0.000, B 0.000, C 0.000 }
gfCNCPoint2[29486] = {X 59.0570, Y 61.0822, Z -3.8333, A 0.000, B 0.000, C 0.000 }
gfCNCPoint2[29487] = {X 57.4323, Y 60.4704, Z -3.8333, A 0.000, B 0.000, C 0.000 }
gfCNCPoint2[29488] = {X 55.8790, Y 59.6950, Z -3.8333, A 0.000, B 0.000, C 0.000 }
gfCNCPoint2[29489] = {X 54.3258, Y 60.4704, Z -3.8333, A 0.000, B 0.000, C 0.000 }
gfCNCPoint2[29490] = {X 52.7011, Y 61.0822, Z -3.8333, A 0.000, B 0.000, C 0.000 }
gfCNCPoint2[29491] = {X 51.0221, Y 61.5238, Z -3.8333, A 0.000, B 0.000, C 0.000 }
gfCNCPoint2[29492] = {X 49.3067, Y 61.7907, Z -3.8333, A 0.000, B 0.000, C 0.000 }
gfCNCPoint2[29493] = {X 47.5729, Y 61.8800, Z -3.8333, A 0.000, B 0.000, C 0.000 }
gfCNCPoint2[29494] = {X 40.6393, Y 61.8800, Z -3.8333, A 0.000, B 0.000, C 0.000 }
gfCNCPoint2[29495] = {X 39.0677, Y 61.8067, Z -3.8333, A 0.000, B 0.000, C 0.000 }
gfCNCPoint2[29496] = {X 37.5098, Y 61.5874, Z -3.8333, A 0.000, B 0.000, C 0.000 }
gfCNCPoint2[29497] = {X 35.9790, Y 61.2239, Z -3.8333, A 0.000, B 0.000, C 0.000 }
gfCNCPoint2[29498] = {X 34.3397, Y 61.9599, Z -3.8333, A 0.000, B 0.000, C 0.000 }
gfCNCPoint2[29499] = {X 32.6439, Y 62.5544, Z -3.8333, A 0.000, B 0.000, C 0.000 }
gfCNCPoint2[29500] = {X 30.9039, Y 63.0033, Z -3.8333, A 0.000, B 0.000, C 0.000 }
gfCNCPoint2[29501] = {X 29.1322, Y 63.3034, Z -3.8333, A 0.000, B 0.000, C 0.000 }
gfCNCPoint2[29502] = {X 27.0258, Y 64.1616, Z -3.8333, A 0.000, B 0.000, C 0.000 }
gfCNCPoint2[29503] = {X 24.8794, Y 64.9145, Z -3.8333, A 0.000, B 0.000, C 0.000 }
gfCNCPoint2[29504] = {X 22.1976, Y 65.6917, Z -3.8333, A 0.000, B 0.000, C 0.000 }
gfCNCPoint2[29505] = {X 19.4677, Y 66.2786, Z -3.8333, A 0.000, B 0.000, C 0.000 }
gfCNCPoint2[29506] = {X 16.7035, Y 66.6724, Z -3.8333, A 0.000, B 0.000, C 0.000 }
gfCNCPoint2[29507] = {X 16.7035, Y 83.2950, Z -3.8333, A 0.000, B 0.000, C 0.000 }
gfCNCPoint2[29508] = {X 111.5046, Y 83.2950, Z -3.8333, A 0.000, B 0.000, C 0.000 }
gfCNCPoint2[29509] = {X 113.0133, Y 81.9631, Z -3.8333, A 0.000, B 0.000, C 0.000 }
gfCNCPoint2[29510] = {X 114.6526, Y 80.7956, Z -3.8333, A 0.000, B 0.000, C 0.000 }
gfCNCPoint2[29511] = {X 116.4046, Y 79.8055, Z -3.8333, A 0.000, B 0.000, C 0.000 }
gfCNCPoint2[29512] = {X 117.4748, Y 81.9537, Z -3.8333, A 0.000, B 0.000, C 0.000 }
gfCNCPoint2[29513] = {X 119.1636, Y 81.2244, Z -3.8333, A 0.000, B 0.000, C 0.000 }
gfCNCPoint2[29514] = {X 120.9217, Y 80.6832, Z -3.8333, A 0.000, B 0.000, C 0.000 }
gfCNCPoint2[29515] = {X 142.4295, Y 57.0646, Z -3.8333, A 0.000, B 0.000, C 0.000 }
gfCNCPoint2[29516] = {X 141.1665, Y 56.9339, Z -3.8333, A 0.000, B 0.000, C 0.000 }
gfCNCPoint2[29517] = {X 139.9241, Y 56.6713, Z -3.8333, A 0.000, B 0.000, C 0.000 }
gfCNCPoint2[29518] = {X 138.7163, Y 56.2798, Z -3.8333, A 0.000, B 0.000, C 0.000 }
gfCNCPoint2[29519] = {X 137.2792, Y 55.6181, Z -3.8333, A 0.000, B 0.000, C 0.000 }
gfCNCPoint2[29520] = {X 135.9409, Y 54.7742, Z -3.8333, A 0.000, B 0.000, C 0.000 }
gfCNCPoint2[29521] = {X 134.7244, Y 53.7626, Z -3.8333, A 0.000, B 0.000, C 0.000 }
gfCNCPoint2[29522] = {X 133.6505, Y 52.6008, Z -3.8333, A 0.000, B 0.000, C 0.000 }
gfCNCPoint2[29523] = {X 132.7377, Y 51.3085, Z -3.8333, A 0.000, B 0.000, C 0.000 }
gfCNCPoint2[29524] = {X 132.0016, Y 49.9080, Z -3.8333, A 0.000, B 0.000, C 0.000 }
gfCNCPoint2[29525] = {X 131.4549, Y 48.4234, Z -3.8333, A 0.000, B 0.000, C 0.000 }
gfCNCPoint2[29526] = {X 131.1845, Y 47.3200, Z -3.8333, A 0.000, B 0.000, C 0.000 }
gfCNCPoint2[29527] = {X 131.0190, Y 46.1961, Z -3.8333, A 0.000, B 0.000, C 0.000 }
gfCNCPoint2[29528] = {X 130.9598, Y 45.0616, Z -3.8333, A 0.000, B 0.000, C 0.000 }
gfCNCPoint2[29529] = {X 130.9601, Y 44.0978, Z -3.8333, A 0.000, B 0.000, C 0.000 }
gfCNCPoint2[29530] = {X 131.0921, Y 42.4244, Z -3.8333, A 0.000, B 0.000, C 0.000 }
gfCNCPoint2[29531] = {X 131.4548, Y 40.7854, Z -3.8333, A 0.000, B 0.000, C 0.000 }
gfCNCPoint2[29532] = {X 133.7565, Y 41.4655, Z -3.8333, A 0.000, B 0.000, C 0.000 }
gfCNCPoint2[29533] = {X 134.2330, Y 40.1906, Z -3.8333, A 0.000, B 0.000, C 0.000 }
gfCNCPoint2[29534] = {X 134.8836, Y 38.9952, Z -3.8333, A 0.000, B 0.000, C 0.000 }
gfCNCPoint2[29535] = {X 134.8836, Y 27.0854, Z -3.8333, A 0.000, B 0.000, C 0.000 }
gfCNCPoint2[29536] = {X 134.3931, Y 27.1259, Z -3.8333, A 0.000, B 0.000, C 0.000 }
gfCNCPoint2[29537] = {X 133.9011, Y 27.1414, Z -3.8333, A 0.000, B 0.000, C 0.000 }
gfCNCPoint2[29538] = {X 133.2006, Y 27.1415, Z -3.8333, A 0.000, B 0.000, C 0.000 }
gfCNCPoint2[29539] = {X 131.9566, Y 27.0613, Z -3.8333, A 0.000, B 0.000, C 0.000 }
gfCNCPoint2[29540] = {X 130.7332, Y 26.8218, Z -3.8333, A 0.000, B 0.000, C 0.000 }
gfCNCPoint2[29541] = {X 129.5508, Y 26.4271, Z -3.8333, A 0.000, B 0.000, C 0.000 }
gfCNCPoint2[29542] = {X 128.4289, Y 25.8837, Z -3.8333, A 0.000, B 0.000, C 0.000 }
gfCNCPoint2[29543] = {X 127.3861, Y 25.2006, Z -3.8333, A 0.000, B 0.000, C 0.000 }
gfCNCPoint2[29544] = {X 126.3452, Y 24.2956, Z -3.8333, A 0.000, B 0.000, C 0.000 }
gfCNCPoint2[29545] = {X 125.4435, Y 23.2519, Z -3.8333, A 0.000, B 0.000, C 0.000 }
gfCNCPoint2[29546] = {X 124.6992, Y 22.0906, Z -3.8333, A 0.000, B 0.000, C 0.000 }
gfCNCPoint2[29547] = {X 124.1276, Y 20.8354, Z -3.8333, A 0.000, B 0.000, C 0.000 }
gfCNCPoint2[29548] = {X 123.7402, Y 19.5116, Z -3.8333, A 0.000, B 0.000, C 0.000 }
gfCNCPoint2[29549] = {X 123.5449, Y 18.1462, Z -3.8333, A 0.000, B 0.000, C 0.000 }
gfCNCPoint2[29550] = {X 123.5438, Y 39.7467, Z -3.8333, A 0.000, B 0.000, C 0.000 }
gfCNCPoint2[29551] = {X 124.1924, Y 40.7407, Z -3.8333, A 0.000, B 0.000, C 0.000 }
gfCNCPoint2[29552] = {X 124.6709, Y 41.8269, Z -3.8333, A 0.000, B 0.000, C 0.000 }
gfCNCPoint2[29553] = {X 124.9665, Y 42.9764, Z -3.8333, A 0.000, B 0.000, C 0.000 }
gfCNCPoint2[29554] = {X 125.0714, Y 44.1587, Z -3.8333, A 0.000, B 0.000, C 0.000 }
gfCNCPoint2[29555] = {X 125.0716, Y 45.0000, Z -3.8333, A 0.000, B 0.000, C 0.000 }
gfCNCPoint2[29556] = {X 124.9610, Y 46.2642, Z -3.8333, A 0.000, B 0.000, C 0.000 }
gfCNCPoint2[29557] = {X 124.6325, Y 47.4899, Z -3.8333, A 0.000, B 0.000, C 0.000 }
gfCNCPoint2[29558] = {X 124.0962, Y 48.6400, Z -3.8333, A 0.000, B 0.000, C 0.000 }
gfCNCPoint2[29559] = {X 123.3684, Y 49.6795, Z -3.8333, A 0.000, B 0.000, C 0.000 }
gfCNCPoint2[29560] = {X 122.4711, Y 50.5768, Z -3.8333, A 0.000, B 0.000, C 0.000 }
gfCNCPoint2[29561] = {X 121.4316, Y 51.3047, Z -3.8333, A 0.000, B 0.000, C 0.000 }
gfCNCPoint2[29562] = {X 120.2815, Y 51.8410, Z -3.8333, A 0.000, B 0.000, C 0.000 }
gfCNCPoint2[29563] = {X 119.0557, Y 52.1694, Z -3.8333, A 0.000, B 0.000, C 0.000 }
gfCNCPoint2[29564] = {X 117.7916, Y 52.2800, Z -3.8333, A 0.000, B 0.000, C 0.000 }
gfCNCPoint2[29565] = {X 111.9185, Y 52.2800, Z -3.8333, A 0.000, B 0.000, C 0.000 }
gfCNCPoint2[29566] = {X 110.8481, Y 52.2009, Z -3.8333, A 0.000, B 0.000, C 0.000 }
gfCNCPoint2[29567] = {X 109.8009, Y 51.9652, Z -3.8333, A 0.000, B 0.000, C 0.000 }
gfCNCPoint2[29568] = {X 108.7998, Y 51.5782, Z -3.8333, A 0.000, B 0.000, C 0.000 }
gfCNCPoint2[29569] = {X 107.8665, Y 51.0481, Z -3.8333, A 0.000, B 0.000, C 0.000 }
gfCNCPoint2[29570] = {X 107.0213, Y 50.3866, Z -3.8333, A 0.000, B 0.000, C 0.000 }
gfCNCPoint2[29571] = {X 106.1743, Y 51.0493, Z -3.8333, A 0.000, B 0.000, C 0.000 }
gfCNCPoint2[29572] = {X 105.2389, Y 51.5800, Z -3.8333, A 0.000, B 0.000, C 0.000 }
gfCNCPoint2[29573] = {X 104.0917, Y 52.0091, Z -3.8333, A 0.000, B 0.000, C 0.000 }
gfCNCPoint2[29574] = {X 102.8887, Y 52.2397, Z -3.8333, A 0.000, B 0.000, C 0.000 }
gfCNCPoint2[29575] = {X 101.6641, Y 52.2655, Z -3.8333, A 0.000, B 0.000, C 0.000 }
gfCNCPoint2[29576] = {X 100.4526, Y 52.0855, Z -3.8333, A 0.000, B 0.000, C 0.000 }
gfCNCPoint2[29577] = {X 99.2883, Y 51.7050, Z -3.8333, A 0.000, B 0.000, C 0.000 }
gfCNCPoint2[29578] = {X 98.2043, Y 51.1347, Z -3.8333, A 0.000, B 0.000, C 0.000 }
gfCNCPoint2[29579] = {X 97.2313, Y 50.3907, Z -3.8333, A 0.000, B 0.000, C 0.000 }
gfCNCPoint2[29580] = {X 96.3865, Y 51.0508, Z -3.8333, A 0.000, B 0.000, C 0.000 }
gfCNCPoint2[29581] = {X 95.4539, Y 51.5797, Z -3.8333, A 0.000, B 0.000, C 0.000 }
gfCNCPoint2[29582] = {X 94.4538, Y 51.9659, Z -3.8333, A 0.000, B 0.000, C 0.000 }
gfCNCPoint2[29583] = {X 93.4078, Y 52.2011, Z -3.8333, A 0.000, B 0.000, C 0.000 }
gfCNCPoint2[29584] = {X 92.3385, Y 52.2800, Z -3.8333, A 0.000, B 0.000, C 0.000 }
gfCNCPoint2[29585] = {X 85.8951, Y 52.2800, Z -3.8333, A 0.000, B 0.000, C 0.000 }
gfCNCPoint2[29586] = {X 84.6852, Y 52.1788, Z -3.8333, A 0.000, B 0.000, C 0.000 }
gfCNCPoint2[29587] = {X 83.5090, Y 51.8779, Z -3.8333, A 0.000, B 0.000, C 0.000 }
gfCNCPoint2[29588] = {X 82.3992, Y 51.3857, Z -3.8333, A 0.000, B 0.000, C 0.000 }
gfCNCPoint2[29589] = {X 81.3866, Y 50.7159, Z -3.8333, A 0.000, B 0.000, C 0.000 }
gfCNCPoint2[29590] = {X 80.5223, Y 52.0937, Z -3.8333, A 0.000, B 0.000, C 0.000 }
gfCNCPoint2[29591] = {X 79.4808, Y 53.3429, Z -3.8333, A 0.000, B 0.000, C 0.000 }
gfCNCPoint2[29592] = {X 78.2809, Y 54.4408, Z -3.8333, A 0.000, B 0.000, C 0.000 }
gfCNCPoint2[29593] = {X 76.9444, Y 55.3676, Z -3.8333, A 0.000, B 0.000, C 0.000 }
gfCNCPoint2[29594] = {X 75.4955, Y 56.1065, Z -3.8333, A 0.000, B 0.000, C 0.000 }
gfCNCPoint2[29595] = {X 73.9605, Y 56.6440, Z -3.8333, A 0.000, B 0.000, C 0.000 }
gfCNCPoint2[29596] = {X 72.3672, Y 56.9705, Z -3.8333, A 0.000, B 0.000, C 0.000 }
gfCNCPoint2[29597] = {X 70.7445, Y 57.0800, Z -3.8333, A 0.000, B 0.000, C 0.000 }
gfCNCPoint2[29598] = {X 64.1851, Y 57.0800, Z -3.8333, A 0.000, B 0.000, C 0.000 }
gfCNCPoint2[29599] = {X 62.6628, Y 56.9837, Z -3.8333, A 0.000, B 0.000, C 0.000 }
gfCNCPoint2[29600] = {X 61.1646, Y 56.6963, Z -3.8333, A 0.000, B 0.000, C 0.000 }
gfCNCPoint2[29601] = {X 59.7147, Y 56.2224, Z -3.8333, A 0.000, B 0.000, C 0.000 }
gfCNCPoint2[29602] = {X 58.3360, Y 55.5695, Z -3.8333, A 0.000, B 0.000, C 0.000 }
gfCNCPoint2[29603] = {X 57.0507, Y 54.7481, Z -3.8333, A 0.000, B 0.000, C 0.000 }
gfCNCPoint2[29604] = {X 55.8790, Y 53.7713, Z -3.8333, A 0.000, B 0.000, C 0.000 }
gfCNCPoint2[29605] = {X 54.7074, Y 54.7481, Z -3.8333, A 0.000, B 0.000, C 0.000 }
gfCNCPoint2[29606] = {X 53.4220, Y 55.5695, Z -3.8333, A 0.000, B 0.000, C 0.000 }
gfCNCPoint2[29607] = {X 52.0434, Y 56.2224, Z -3.8333, A 0.000, B 0.000, C 0.000 }
gfCNCPoint2[29608] = {X 50.5934, Y 56.6963, Z -3.8333, A 0.000, B 0.000, C 0.000 }
gfCNCPoint2[29609] = {X 49.0953, Y 56.9837, Z -3.8333, A 0.000, B 0.000, C 0.000 }
gfCNCPoint2[29610] = {X 47.5729, Y 57.0800, Z -3.8333, A 0.000, B 0.000, C 0.000 }
gfCNCPoint2[29611] = {X 40.6393, Y 57.0800, Z -3.8333, A 0.000, B 0.000, C 0.000 }
gfCNCPoint2[29612] = {X 39.3237, Y 57.0082, Z -3.8333, A 0.000, B 0.000, C 0.000 }
gfCNCPoint2[29613] = {X 38.0238, Y 56.7935, Z -3.8333, A 0.000, B 0.000, C 0.000 }
gfCNCPoint2[29614] = {X 36.7550, Y 56.4385, Z -3.8333, A 0.000, B 0.000, C 0.000 }
gfCNCPoint2[29615] = {X 35.5324, Y 55.9474, Z -3.8333, A 0.000, B 0.000, C 0.000 }
gfCNCPoint2[29616] = {X 34.1217, Y 56.7822, Z -3.8333, A 0.000, B 0.000, C 0.000 }
gfCNCPoint2[29617] = {X 32.6346, Y 57.4720, Z -3.8333, A 0.000, B 0.000, C 0.000 }
gfCNCPoint2[29618] = {X 31.0862, Y 58.0101, Z -3.8333, A 0.000, B 0.000, C 0.000 }
gfCNCPoint2[29619] = {X 29.4919, Y 58.3911, Z -3.8333, A 0.000, B 0.000, C 0.000 }
gfCNCPoint2[29620] = {X 27.8675, Y 58.6111, Z -3.8333, A 0.000, B 0.000, C 0.000 }
gfCNCPoint2[29621] = {X 25.6555, Y 59.5462, Z -3.8333, A 0.000, B 0.000, C 0.000 }
gfCNCPoint2[29622] = {X 23.3927, Y 60.3505, Z -3.8333, A 0.000, B 0.000, C 0.000 }
gfCNCPoint2[29623] = {X 21.1518, Y 61.0049, Z -3.8333, A 0.000, B 0.000, C 0.000 }
gfCNCPoint2[29624] = {X 18.8722, Y 61.5081, Z -3.8333, A 0.000, B 0.000, C 0.000 }
gfCNCPoint2[29625] = {X 16.5640, Y 61.8580, Z -3.8333, A 0.000, B 0.000, C 0.000 }
gfCNCPoint2[29626] = {X 14.2376, Y 62.0529, Z -3.8333, A 0.000, B 0.000, C 0.000 }
gfCNCPoint2[29627] = {X 11.9035, Y 62.0920, Z -3.8333, A 0.000, B 0.000, C 0.000 }
gfCNCPoint2[29628] = {X 11.9035, Y 88.0950, Z -3.8333, A 0.000, B 0.000, C 0.000 }
gfCNCPoint2[29629] = {X 113.6327, Y 88.0950, Z -3.8333, A 0.000, B 0.000, C 0.000 }
gfCNCPoint2[29630] = {X 114.7662, Y 86.8202, Z -3.8333, A 0.000, B 0.000, C 0.000 }
gfCNCPoint2[29631] = {X 116.0418, Y 85.6876, Z -3.8333, A 0.000, B 0.000, C 0.000 }
gfCNCPoint2[29632] = {X 117.4417, Y 84.7128, Z -3.8333, A 0.000, B 0.000, C 0.000 }
gfCNCPoint2[29633] = {X 118.9465, Y 83.9095, Z -3.8333, A 0.000, B 0.000, C 0.000 }
gfCNCPoint2[29634] = {X 120.5354, Y 83.2887, Z -3.8333, A 0.000, B 0.000, C 0.000 }
gfCNCPoint2[29635] = {X 122.1863, Y 82.8590, Z -3.8333, A 0.000, B 0.000, C 0.000 }
gfCNCPoint2[29636] = {X 144.8180, Y 58.0062, Z -3.8333, A 0.000, B 0.000, C 0.000 }
gfCNCPoint2[29637] = {X 144.9144, Y 56.3319, Z -3.8333, A 0.000, B 0.000, C 0.000 }
gfCNCPoint2[29638] = {X 145.2037, Y 54.6800, Z -3.8333, A 0.000, B 0.000, C 0.000 }
gfCNCPoint2[29639] = {X 143.0396, Y 54.6800, Z -3.8333, A 0.000, B 0.000, C 0.000 }
gfCNCPoint2[29640] = {X 142.7951, Y 54.6769, Z -3.8333, A 0.000, B 0.000, C 0.000 }
gfCNCPoint2[29641] = {X 142.5507, Y 54.6676, Z -3.8333, A 0.000, B 0.000, C 0.000 }
gfCNCPoint2[29642] = {X 141.0976, Y 54.4832, Z -3.8333, A 0.000, B 0.000, C 0.000 }
gfCNCPoint2[29643] = {X 139.6891, Y 54.0816, Z -3.8333, A 0.000, B 0.000, C 0.000 }
gfCNCPoint2[29644] = {X 138.3572, Y 53.4722, Z -3.8333, A 0.000, B 0.000, C 0.000 }
gfCNCPoint2[29645] = {X 137.1325, Y 52.6687, Z -3.8333, A 0.000, B 0.000, C 0.000 }
gfCNCPoint2[29646] = {X 136.0431, Y 51.6897, Z -3.8333, A 0.000, B 0.000, C 0.000 }
gfCNCPoint2[29647] = {X 135.1139, Y 50.5575, Z -3.8333, A 0.000, B 0.000, C 0.000 }
gfCNCPoint2[29648] = {X 134.3661, Y 49.2980, Z -3.8333, A 0.000, B 0.000, C 0.000 }
gfCNCPoint2[29649] = {X 133.8169, Y 47.9402, Z -3.8333, A 0.000, B 0.000, C 0.000 }
gfCNCPoint2[29650] = {X 133.4789, Y 46.5150, Z -3.8333, A 0.000, B 0.000, C 0.000 }
gfCNCPoint2[29651] = {X 133.3598, Y 45.0552, Z -3.8333, A 0.000, B 0.000, C 0.000 }
gfCNCPoint2[29652] = {X 133.3601, Y 44.1104, Z -3.8333, A 0.000, B 0.000, C 0.000 }
gfCNCPoint2[29653] = {X 133.4665, Y 42.7742, Z -3.8333, A 0.000, B 0.000, C 0.000 }
gfCNCPoint2[29654] = {X 133.7565, Y 41.4655, Z -3.8333, A 0.000, B 0.000, C 0.000 }
gfCNCPoint2[29655] = {X 136.0581, Y 42.1457, Z -3.8333, A 0.000, B 0.000, C 0.000 }
gfCNCPoint2[29656] = {X 136.3664, Y 41.2990, Z -3.8333, A 0.000, B 0.000, C 0.000 }
gfCNCPoint2[29657] = {X 136.7770, Y 40.4969, Z -3.8333, A 0.000, B 0.000, C 0.000 }
gfCNCPoint2[29658] = {X 137.2836, Y 39.7516, Z -3.8333, A 0.000, B 0.000, C 0.000 }
gfCNCPoint2[29659] = {X 137.2836, Y 23.8768, Z -3.8333, A 0.000, B 0.000, C 0.000 }
gfCNCPoint2[29660] = {X 136.4352, Y 24.2641, Z -3.8333, A 0.000, B 0.000, C 0.000 }
gfCNCPoint2[29661] = {X 135.5443, Y 24.5398, Z -3.8333, A 0.000, B 0.000, C 0.000 }
gfCNCPoint2[29662] = {X 134.6254, Y 24.6993, Z -3.8333, A 0.000, B 0.000, C 0.000 }
gfCNCPoint2[29663] = {X 134.2595, Y 24.7296, Z -3.8333, A 0.000, B 0.000, C 0.000 }
gfCNCPoint2[29664] = {X 133.8926, Y 24.7414, Z -3.8333, A 0.000, B 0.000, C 0.000 }
gfCNCPoint2[29665] = {X 133.2006, Y 24.7415, Z -3.8333, A 0.000, B 0.000, C 0.000 }
gfCNCPoint2[29666] = {X 131.9929, Y 24.6407, Z -3.8333, A 0.000, B 0.000, C 0.000 }
gfCNCPoint2[29667] = {X 130.8187, Y 24.3408, Z -3.8333, A 0.000, B 0.000, C 0.000 }
gfCNCPoint2[29668] = {X 129.7104, Y 23.8503, Z -3.8333, A 0.000, B 0.000, C 0.000 }
gfCNCPoint2[29669] = {X 128.6989, Y 23.1828, Z -3.8333, A 0.000, B 0.000, C 0.000 }
gfCNCPoint2[29670] = {X 127.8121, Y 22.3567, Z -3.8333, A 0.000, B 0.000, C 0.000 }
gfCNCPoint2[29671] = {X 127.0747, Y 21.3949, Z -3.8333, A 0.000, B 0.000, C 0.000 }
gfCNCPoint2[29672] = {X 126.5071, Y 20.3242, Z -3.8333, A 0.000, B 0.000, C 0.000 }
gfCNCPoint2[29673] = {X 126.1249, Y 19.1740, Z -3.8333, A 0.000, B 0.000, C 0.000 }
gfCNCPoint2[29674] = {X 125.9389, Y 17.9765, Z -3.8333, A 0.000, B 0.000, C 0.000 }
gfCNCPoint2[29675] = {X 125.9252, Y 17.7192, Z -3.8333, A 0.000, B 0.000, C 0.000 }
gfCNCPoint2[29676] = {X 125.9206, Y 17.4615, Z -3.8333, A 0.000, B 0.000, C 0.000 }
gfCNCPoint2[29677] = {X 125.9206, Y 10.4835, Z -3.8333, A 0.000, B 0.000, C 0.000 }
gfCNCPoint2[29678] = {X 125.9372, Y 9.9931, Z -3.8333, A 0.000, B 0.000, C 0.000 }
gfCNCPoint2[29679] = {X 125.9867, Y 9.5050, Z -3.8333, A 0.000, B 0.000, C 0.000 }
gfCNCPoint2[29680] = {X 121.8686, Y 9.5050, Z -3.8333, A 0.000, B 0.000, C 0.000 }
gfCNCPoint2[29681] = {X 122.3090, Y 10.3410, Z -3.8333, A 0.000, B 0.000, C 0.000 }
gfCNCPoint2[29682] = {X 122.5801, Y 11.2463, Z -3.8333, A 0.000, B 0.000, C 0.000 }
gfCNCPoint2[29683] = {X 122.6716, Y 12.1868, Z -3.8333, A 0.000, B 0.000, C 0.000 }
gfCNCPoint2[29684] = {X 122.6714, Y 13.0237, Z -3.8333, A 0.000, B 0.000, C 0.000 }
gfCNCPoint2[29685] = {X 122.5640, Y 13.9969, Z -3.8333, A 0.000, B 0.000, C 0.000 }
gfCNCPoint2[29686] = {X 122.2646, Y 14.9290, Z -3.8333, A 0.000, B 0.000, C 0.000 }
gfCNCPoint2[29687] = {X 121.7852, Y 15.7826, Z -3.8333, A 0.000, B 0.000, C 0.000 }
gfCNCPoint2[29688] = {X 121.1450, Y 16.5233, Z -3.8333, A 0.000, B 0.000, C 0.000 }
gfCNCPoint2[29689] = {X 121.1438, Y 40.6624, Z -3.8333, A 0.000, B 0.000, C 0.000 }
gfCNCPoint2[29690] = {X 121.7853, Y 41.4044, Z -3.8333, A 0.000, B 0.000, C 0.000 }
gfCNCPoint2[29691] = {X 122.2654, Y 42.2597, Z -3.8333, A 0.000, B 0.000, C 0.000 }
gfCNCPoint2[29692] = {X 122.5648, Y 43.1937, Z -3.8333, A 0.000, B 0.000, C 0.000 }
gfCNCPoint2[29693] = {X 122.6714, Y 44.1688, Z -3.8333, A 0.000, B 0.000, C 0.000 }
gfCNCPoint2[29694] = {X 122.6716, Y 45.0000, Z -3.8333, A 0.000, B 0.000, C 0.000 }
gfCNCPoint2[29695] = {X 122.5778, Y 45.9520, Z -3.8333, A 0.000, B 0.000, C 0.000 }
gfCNCPoint2[29696] = {X 122.3001, Y 46.8675, Z -3.8333, A 0.000, B 0.000, C 0.000 }
gfCNCPoint2[29697] = {X 121.8491, Y 47.7112, Z -3.8333, A 0.000, B 0.000, C 0.000 }
gfCNCPoint2[29698] = {X 121.2423, Y 48.4507, Z -3.8333, A 0.000, B 0.000, C 0.000 }
gfCNCPoint2[29699] = {X 120.5028, Y 49.0576, Z -3.8333, A 0.000, B 0.000, C 0.000 }
gfCNCPoint2[29700] = {X 119.6591, Y 49.5085, Z -3.8333, A 0.000, B 0.000, C 0.000 }
gfCNCPoint2[29701] = {X 118.7436, Y 49.7862, Z -3.8333, A 0.000, B 0.000, C 0.000 }
gfCNCPoint2[29702] = {X 117.7916, Y 49.8800, Z -3.8333, A 0.000, B 0.000, C 0.000 }
gfCNCPoint2[29703] = {X 111.9185, Y 49.8800, Z -3.8333, A 0.000, B 0.000, C 0.000 }
gfCNCPoint2[29704] = {X 111.0234, Y 49.7972, Z -3.8333, A 0.000, B 0.000, C 0.000 }
gfCNCPoint2[29705] = {X 110.1587, Y 49.5517, Z -3.8333, A 0.000, B 0.000, C 0.000 }
gfCNCPoint2[29706] = {X 109.3537, Y 49.1517, Z -3.8333, A 0.000, B 0.000, C 0.000 }
gfCNCPoint2[29707] = {X 108.6357, Y 48.6108, Z -3.8333, A 0.000, B 0.000, C 0.000 }
gfCNCPoint2[29708] = {X 108.0714, Y 48.0024, Z -3.8333, A 0.000, B 0.000, C 0.000 }
gfCNCPoint2[29709] = {X 107.6183, Y 47.3071, Z -3.8333, A 0.000, B 0.000, C 0.000 }
gfCNCPoint2[29710] = {X 107.2895, Y 46.5451, Z -3.8333, A 0.000, B 0.000, C 0.000 }
gfCNCPoint2[29711] = {X 107.0947, Y 45.7384, Z -3.8333, A 0.000, B 0.000, C 0.000 }
gfCNCPoint2[29712] = {X 106.6287, Y 46.8769, Z -3.8333, A 0.000, B 0.000, C 0.000 }
gfCNCPoint2[29713] = {X 106.1131, Y 47.8110, Z -3.8333, A 0.000, B 0.000, C 0.000 }
gfCNCPoint2[29714] = {X 105.4068, Y 48.6108, Z -3.8333, A 0.000, B 0.000, C 0.000 }
gfCNCPoint2[29715] = {X 104.8391, Y 49.0550, Z -3.8333, A 0.000, B 0.000, C 0.000 }
gfCNCPoint2[29716] = {X 104.2121, Y 49.4107, Z -3.8333, A 0.000, B 0.000, C 0.000 }
gfCNCPoint2[29717] = {X 103.3106, Y 49.7335, Z -3.8333, A 0.000, B 0.000, C 0.000 }
gfCNCPoint2[29718] = {X 102.3635, Y 49.8741, Z -3.8333, A 0.000, B 0.000, C 0.000 }
gfCNCPoint2[29719] = {X 101.4071, Y 49.8271, Z -3.8333, A 0.000, B 0.000, C 0.000 }
gfCNCPoint2[29720] = {X 100.4784, Y 49.5941, Z -3.8333, A 0.000, B 0.000, C 0.000 }
gfCNCPoint2[29721] = {X 99.6130, Y 49.1844, Z -3.8333, A 0.000, B 0.000, C 0.000 }
gfCNCPoint2[29722] = {X 98.8443, Y 48.6135, Z -3.8333, A 0.000, B 0.000, C 0.000 }
gfCNCPoint2[29723] = {X 98.1362, Y 47.8127, Z -3.8333, A 0.000, B 0.000, C 0.000 }
gfCNCPoint2[29724] = {X 97.6194, Y 46.8769, Z -3.8333, A 0.000, B 0.000, C 0.000 }
gfCNCPoint2[29725] = {X 97.1600, Y 45.7536, Z -3.8333, A 0.000, B 0.000, C 0.000 }
gfCNCPoint2[29726] = {X 96.9635, Y 46.5570, Z -3.8333, A 0.000, B 0.000, C 0.000 }
gfCNCPoint2[29727] = {X 96.6342, Y 47.3156, Z -3.8333, A 0.000, B 0.000, C 0.000 }
gfCNCPoint2[29728] = {X 96.1814, Y 48.0078, Z -3.8333, A 0.000, B 0.000, C 0.000 }
gfCNCPoint2[29729] = {X 95.6183, Y 48.6135, Z -3.8333, A 0.000, B 0.000, C 0.000 }
gfCNCPoint2[29730] = {X 94.9007, Y 49.1533, Z -3.8333, A 0.000, B 0.000, C 0.000 }
gfCNCPoint2[29731] = {X 94.0964, Y 49.5524, Z -3.8333, A 0.000, B 0.000, C 0.000 }
gfCNCPoint2[29732] = {X 93.2326, Y 49.7974, Z -3.8333, A 0.000, B 0.000, C 0.000 }
gfCNCPoint2[29733] = {X 92.3385, Y 49.8800, Z -3.8333, A 0.000, B 0.000, C 0.000 }
gfCNCPoint2[29734] = {X 85.8951, Y 49.8800, Z -3.8333, A 0.000, B 0.000, C 0.000 }
gfCNCPoint2[29735] = {X 85.0841, Y 49.8121, Z -3.8333, A 0.000, B 0.000, C 0.000 }
gfCNCPoint2[29736] = {X 84.2956, Y 49.6104, Z -3.8333, A 0.000, B 0.000, C 0.000 }
gfCNCPoint2[29737] = {X 83.5517, Y 49.2805, Z -3.8333, A 0.000, B 0.000, C 0.000 }
gfCNCPoint2[29738] = {X 82.8729, Y 48.8316, Z -3.8333, A 0.000, B 0.000, C 0.000 }
gfCNCPoint2[29739] = {X 82.2391, Y 48.2324, Z -3.8333, A 0.000, B 0.000, C 0.000 }
gfCNCPoint2[29740] = {X 81.7221, Y 47.5300, Z -3.8333, A 0.000, B 0.000, C 0.000 }
gfCNCPoint2[29741] = {X 81.3384, Y 46.7467, Z -3.8333, A 0.000, B 0.000, C 0.000 }
gfCNCPoint2[29742] = {X 81.1002, Y 45.9077, Z -3.8333, A 0.000, B 0.000, C 0.000 }
gfCNCPoint2[29743] = {X 81.0152, Y 45.0397, Z -3.8333, A 0.000, B 0.000, C 0.000 }
gfCNCPoint2[29744] = {X 81.0151, Y 44.2035, Z -3.8333, A 0.000, B 0.000, C 0.000 }
gfCNCPoint2[29745] = {X 81.1201, Y 43.2199, Z -3.8333, A 0.000, B 0.000, C 0.000 }
gfCNCPoint2[29746] = {X 81.4189, Y 42.2769, Z -3.8333, A 0.000, B 0.000, C 0.000 }
gfCNCPoint2[29747] = {X 81.8997, Y 41.4124, Z -3.8333, A 0.000, B 0.000, C 0.000 }
gfCNCPoint2[29748] = {X 82.5431, Y 40.6610, Z -3.8333, A 0.000, B 0.000, C 0.000 }
gfCNCPoint2[29749] = {X 82.5428, Y 16.5244, Z -3.8333, A 0.000, B 0.000, C 0.000 }
gfCNCPoint2[29750] = {X 81.9016, Y 15.7827, Z -3.8333, A 0.000, B 0.000, C 0.000 }
gfCNCPoint2[29751] = {X 81.4215, Y 14.9278, Z -3.8333, A 0.000, B 0.000, C 0.000 }
gfCNCPoint2[29752] = {X 81.1221, Y 13.9942, Z -3.8333, A 0.000, B 0.000, C 0.000 }
gfCNCPoint2[29753] = {X 81.0153, Y 13.0196, Z -3.8333, A 0.000, B 0.000, C 0.000 }
gfCNCPoint2[29754] = {X 81.0151, Y 12.1868, Z -3.8333, A 0.000, B 0.000, C 0.000 }
gfCNCPoint2[29755] = {X 81.0160, Y 12.0923, Z -3.8333, A 0.000, B 0.000, C 0.000 }
gfCNCPoint2[29756] = {X 81.0187, Y 11.9979, Z -3.8333, A 0.000, B 0.000, C 0.000 }
gfCNCPoint2[29757] = {X 81.1324, Y 11.1230, Z -3.8333, A 0.000, B 0.000, C 0.000 }
gfCNCPoint2[29758] = {X 81.4018, Y 10.2829, Z -3.8333, A 0.000, B 0.000, C 0.000 }
gfCNCPoint2[29759] = {X 81.8180, Y 9.5050, Z -3.8333, A 0.000, B 0.000, C 0.000 }
gfCNCPoint2[29760] = {X 82.2190, Y 9.7688, Z -3.8333, A 0.000, B 0.000, C 0.000 }
gfCNCPoint2[29761] = {X 82.7659, Y 9.0936, Z -3.8333, A 0.000, B 0.000, C 0.000 }
gfCNCPoint2[29762] = {X 83.4347, Y 8.5390, Z -3.8333, A 0.000, B 0.000, C 0.000 }
gfCNCPoint2[29763] = {X 84.1995, Y 8.1266, Z -3.8333, A 0.000, B 0.000, C 0.000 }
gfCNCPoint2[29764] = {X 85.0304, Y 7.8726, Z -3.8333, A 0.000, B 0.000, C 0.000 }
gfCNCPoint2[29765] = {X 85.8951, Y 7.7868, Z -3.8333, A 0.000, B 0.000, C 0.000 }
gfCNCPoint2[29766] = {X 94.0497, Y 7.7868, Z -3.8333, A 0.000, B 0.000, C 0.000 }
gfCNCPoint2[29767] = {X 95.0288, Y 7.8971, Z -3.8333, A 0.000, B 0.000, C 0.000 }
gfCNCPoint2[29768] = {X 95.9588, Y 8.2226, Z -3.8333, A 0.000, B 0.000, C 0.000 }
gfCNCPoint2[29769] = {X 96.7930, Y 8.7468, Z -3.8333, A 0.000, B 0.000, C 0.000 }
gfCNCPoint2[29770] = {X 97.4897, Y 9.4435, Z -3.8333, A 0.000, B 0.000, C 0.000 }
gfCNCPoint2[29771] = {X 98.0139, Y 10.2777, Z -3.8333, A 0.000, B 0.000, C 0.000 }
gfCNCPoint2[29772] = {X 98.3394, Y 11.2077, Z -3.8333, A 0.000, B 0.000, C 0.000 }
gfCNCPoint2[29773] = {X 98.4497, Y 12.1868, Z -3.8333, A 0.000, B 0.000, C 0.000 }
gfCNCPoint2[29774] = {X 98.4494, Y 13.0233, Z -3.8333, A 0.000, B 0.000, C 0.000 }
gfCNCPoint2[29775] = {X 98.3724, Y 13.7993, Z -3.8333, A 0.000, B 0.000, C 0.000 }
gfCNCPoint2[29776] = {X 98.1595, Y 14.5494, Z -3.8333, A 0.000, B 0.000, C 0.000 }
gfCNCPoint2[29777] = {X 97.8176, Y 15.2502, Z -3.8333, A 0.000, B 0.000, C 0.000 }
gfCNCPoint2[29778] = {X 98.3675, Y 16.6194, Z -3.8333, A 0.000, B 0.000, C 0.000 }
gfCNCPoint2[29779] = {X 101.8765, Y 25.3175, Z -3.8333, A 0.000, B 0.000, C 0.000 }
gfCNCPoint2[29780] = {X 105.9242, Y 15.2232, Z -3.8333, A 0.000, B 0.000, C 0.000 }
gfCNCPoint2[29781] = {X 105.5857, Y 14.5156, Z -3.8333, A 0.000, B 0.000, C 0.000 }
gfCNCPoint2[29782] = {X 105.3782, Y 13.7592, Z -3.8333, A 0.000, B 0.000, C 0.000 }
gfCNCPoint2[29783] = {X 105.3083, Y 12.9779, Z -3.8333, A 0.000, B 0.000, C 0.000 }
gfCNCPoint2[29784] = {X 105.3083, Y 12.1868, Z -3.8333, A 0.000, B 0.000, C 0.000 }
gfCNCPoint2[29785] = {X 105.4186, Y 11.2077, Z -3.8333, A 0.000, B 0.000, C 0.000 }
gfCNCPoint2[29786] = {X 105.7440, Y 10.2777, Z -3.8333, A 0.000, B 0.000, C 0.000 }
gfCNCPoint2[29787] = {X 106.2682, Y 9.4435, Z -3.8333, A 0.000, B 0.000, C 0.000 }
gfCNCPoint2[29788] = {X 106.9649, Y 8.7468, Z -3.8333, A 0.000, B 0.000, C 0.000 }
gfCNCPoint2[29789] = {X 107.7992, Y 8.2226, Z -3.8333, A 0.000, B 0.000, C 0.000 }
gfCNCPoint2[29790] = {X 108.7292, Y 7.8971, Z -3.8333, A 0.000, B 0.000, C 0.000 }
gfCNCPoint2[29791] = {X 109.7083, Y 7.7868, Z -3.8333, A 0.000, B 0.000, C 0.000 }
gfCNCPoint2[29792] = {X 117.7916, Y 7.7868, Z -3.8333, A 0.000, B 0.000, C 0.000 }
gfCNCPoint2[29793] = {X 118.7707, Y 7.8971, Z -3.8333, A 0.000, B 0.000, C 0.000 }
gfCNCPoint2[29794] = {X 119.7007, Y 8.2226, Z -3.8333, A 0.000, B 0.000, C 0.000 }
gfCNCPoint2[29795] = {X 120.5349, Y 8.7468, Z -3.8333, A 0.000, B 0.000, C 0.000 }
gfCNCPoint2[29796] = {X 121.2316, Y 9.4435, Z -3.8333, A 0.000, B 0.000, C 0.000 }
gfCNCPoint2[29797] = {X 121.7558, Y 10.2777, Z -3.8333, A 0.000, B 0.000, C 0.000 }
gfCNCPoint2[29798] = {X 122.0813, Y 11.2077, Z -3.8333, A 0.000, B 0.000, C 0.000 }
gfCNCPoint2[29799] = {X 122.1916, Y 12.1868, Z -3.8333, A 0.000, B 0.000, C 0.000 }
gfCNCPoint2[29800] = {X 122.1913, Y 13.0233, Z -3.8333, A 0.000, B 0.000, C 0.000 }
gfCNCPoint2[29801] = {X 122.0831, Y 13.9490, Z -3.8333, A 0.000, B 0.000, C 0.000 }
gfCNCPoint2[29802] = {X 121.7823, Y 14.8312, Z -3.8333, A 0.000, B 0.000, C 0.000 }
gfCNCPoint2[29803] = {X 121.3024, Y 15.6302, Z -3.8333, A 0.000, B 0.000, C 0.000 }
gfCNCPoint2[29804] = {X 120.6650, Y 16.3102, Z -3.8333, A 0.000, B 0.000, C 0.000 }
gfCNCPoint2[29805] = {X 120.6638, Y 40.8760, Z -3.8333, A 0.000, B 0.000, C 0.000 }
gfCNCPoint2[29806] = {X 120.6784, Y 40.8882, Z -3.8333, A 0.000, B 0.000, C 0.000 }
gfCNCPoint2[29807] = {X 121.3172, Y 41.5763, Z -3.8333, A 0.000, B 0.000, C 0.000 }
gfCNCPoint2[29808] = {X 121.7955, Y 42.3843, Z -3.8333, A 0.000, B 0.000, C 0.000 }
gfCNCPoint2[29809] = {X 122.0914, Y 43.2754, Z -3.8333, A 0.000, B 0.000, C 0.000 }
gfCNCPoint2[29810] = {X 122.1916, Y 44.2089, Z -3.8333, A 0.000, B 0.000, C 0.000 }
gfCNCPoint2[29811] = {X 122.1916, Y 45.0000, Z -3.8333, A 0.000, B 0.000, C 0.000 }
gfCNCPoint2[29812] = {X 122.0813, Y 45.9791, Z -3.8333, A 0.000, B 0.000, C 0.000 }
gfCNCPoint2[29813] = {X 121.7558, Y 46.9091, Z -3.8333, A 0.000, B 0.000, C 0.000 }
gfCNCPoint2[29814] = {X 121.2316, Y 47.7434, Z -3.8333, A 0.000, B 0.000, C 0.000 }
gfCNCPoint2[29815] = {X 120.5349, Y 48.4401, Z -3.8333, A 0.000, B 0.000, C 0.000 }
gfCNCPoint2[29816] = {X 119.7007, Y 48.9643, Z -3.8333, A 0.000, B 0.000, C 0.000 }
gfCNCPoint2[29817] = {X 118.7707, Y 49.2897, Z -3.8333, A 0.000, B 0.000, C 0.000 }
gfCNCPoint2[29818] = {X 117.7916, Y 49.4000, Z -3.8333, A 0.000, B 0.000, C 0.000 }
gfCNCPoint2[29819] = {X 111.9185, Y 49.4000, Z -3.8333, A 0.000, B 0.000, C 0.000 }
gfCNCPoint2[29820] = {X 110.9394, Y 49.2897, Z -3.8333, A 0.000, B 0.000, C 0.000 }
gfCNCPoint2[29821] = {X 110.0094, Y 48.9643, Z -3.8333, A 0.000, B 0.000, C 0.000 }
gfCNCPoint2[29822] = {X 109.1751, Y 48.4400, Z -3.8333, A 0.000, B 0.000, C 0.000 }
gfCNCPoint2[29823] = {X 108.4784, Y 47.7433, Z -3.8333, A 0.000, B 0.000, C 0.000 }
gfCNCPoint2[29824] = {X 107.9542, Y 46.9091, Z -3.8333, A 0.000, B 0.000, C 0.000 }
gfCNCPoint2[29825] = {X 107.6288, Y 45.9791, Z -3.8333, A 0.000, B 0.000, C 0.000 }
gfCNCPoint2[29826] = {X 107.5185, Y 45.0000, Z -3.8333, A 0.000, B 0.000, C 0.000 }
gfCNCPoint2[29827] = {X 107.5185, Y 44.1793, Z -3.8333, A 0.000, B 0.000, C 0.000 }
gfCNCPoint2[29828] = {X 107.5549, Y 43.6254, Z -3.8333, A 0.000, B 0.000, C 0.000 }
gfCNCPoint2[29829] = {X 107.6635, Y 43.0809, Z -3.8333, A 0.000, B 0.000, C 0.000 }
gfCNCPoint2[29830] = {X 106.1856, Y 46.6923, Z -3.8333, A 0.000, B 0.000, C 0.000 }
gfCNCPoint2[29831] = {X 105.8087, Y 47.4049, Z -3.8333, A 0.000, B 0.000, C 0.000 }
gfCNCPoint2[29832] = {X 105.3081, Y 48.0367, Z -3.8333, A 0.000, B 0.000, C 0.000 }
gfCNCPoint2[29833] = {X 104.7006, Y 48.5667, Z -3.8333, A 0.000, B 0.000, C 0.000 }
gfCNCPoint2[29834] = {X 104.0067, Y 48.9769, Z -3.8333, A 0.000, B 0.000, C 0.000 }
gfCNCPoint2[29835] = {X 103.0414, Y 49.3033, Z -3.8333, A 0.000, B 0.000, C 0.000 }
gfCNCPoint2[29836] = {X 102.0269, Y 49.3989, Z -3.8333, A 0.000, B 0.000, C 0.000 }
gfCNCPoint2[29837] = {X 101.0176, Y 49.2586, Z -3.8333, A 0.000, B 0.000, C 0.000 }
gfCNCPoint2[29838] = {X 100.0676, Y 48.8899, Z -3.8333, A 0.000, B 0.000, C 0.000 }
gfCNCPoint2[29839] = {X 99.2280, Y 48.3125, Z -3.8333, A 0.000, B 0.000, C 0.000 }
gfCNCPoint2[29840] = {X 98.5436, Y 47.5575, Z -3.8333, A 0.000, B 0.000, C 0.000 }
gfCNCPoint2[29841] = {X 98.0514, Y 46.6653, Z -3.8333, A 0.000, B 0.000, C 0.000 }
gfCNCPoint2[29842] = {X 96.5867, Y 43.0833, Z -3.8333, A 0.000, B 0.000, C 0.000 }
gfCNCPoint2[29843] = {X 96.6984, Y 43.6413, Z -3.8333, A 0.000, B 0.000, C 0.000 }
gfCNCPoint2[29844] = {X 96.7385, Y 44.2089, Z -3.8333, A 0.000, B 0.000, C 0.000 }
gfCNCPoint2[29845] = {X 96.7383, Y 45.0423, Z -3.8333, A 0.000, B 0.000, C 0.000 }
gfCNCPoint2[29846] = {X 96.6200, Y 46.0144, Z -3.8333, A 0.000, B 0.000, C 0.000 }
gfCNCPoint2[29847] = {X 96.2896, Y 46.9363, Z -3.8333, A 0.000, B 0.000, C 0.000 }
gfCNCPoint2[29848] = {X 95.7635, Y 47.7622, Z -3.8333, A 0.000, B 0.000, C 0.000 }
gfCNCPoint2[29849] = {X 95.0677, Y 48.4513, Z -3.8333, A 0.000, B 0.000, C 0.000 }
gfCNCPoint2[29850] = {X 94.2367, Y 48.9695, Z -3.8333, A 0.000, B 0.000, C 0.000 }
gfCNCPoint2[29851] = {X 93.3117, Y 49.2910, Z -3.8333, A 0.000, B 0.000, C 0.000 }
gfCNCPoint2[29852] = {X 92.3385, Y 49.4000, Z -3.8333, A 0.000, B 0.000, C 0.000 }
gfCNCPoint2[29853] = {X 85.8951, Y 49.4000, Z -3.8333, A 0.000, B 0.000, C 0.000 }
gfCNCPoint2[29854] = {X 84.9160, Y 49.2897, Z -3.8333, A 0.000, B 0.000, C 0.000 }
gfCNCPoint2[29855] = {X 83.9860, Y 48.9643, Z -3.8333, A 0.000, B 0.000, C 0.000 }
gfCNCPoint2[29856] = {X 83.1517, Y 48.4400, Z -3.8333, A 0.000, B 0.000, C 0.000 }
gfCNCPoint2[29857] = {X 82.4550, Y 47.7433, Z -3.8333, A 0.000, B 0.000, C 0.000 }
gfCNCPoint2[29858] = {X 81.9308, Y 46.9091, Z -3.8333, A 0.000, B 0.000, C 0.000 }
gfCNCPoint2[29859] = {X 81.6054, Y 45.9791, Z -3.8333, A 0.000, B 0.000, C 0.000 }
gfCNCPoint2[29860] = {X 81.4951, Y 45.0000, Z -3.8333, A 0.000, B 0.000, C 0.000 }
gfCNCPoint2[29861] = {X 81.4951, Y 44.2065, Z -3.8333, A 0.000, B 0.000, C 0.000 }
gfCNCPoint2[29862] = {X 81.6004, Y 43.2693, Z -3.8333, A 0.000, B 0.000, C 0.000 }
gfCNCPoint2[29863] = {X 81.9005, Y 42.3752, Z -3.8333, A 0.000, B 0.000, C 0.000 }
gfCNCPoint2[29864] = {X 82.3819, Y 41.5642, Z -3.8333, A 0.000, B 0.000, C 0.000 }
gfCNCPoint2[29865] = {X 83.0231, Y 40.8726, Z -3.8333, A 0.000, B 0.000, C 0.000 }
gfCNCPoint2[29866] = {X 83.0228, Y 16.3112, Z -3.8333, A 0.000, B 0.000, C 0.000 }
gfCNCPoint2[29867] = {X 82.3781, Y 15.6221, Z -3.8333, A 0.000, B 0.000, C 0.000 }
gfCNCPoint2[29868] = {X 81.8952, Y 14.8113, Z -3.8333, A 0.000, B 0.000, C 0.000 }
gfCNCPoint2[29869] = {X 81.5963, Y 13.9162, Z -3.8333, A 0.000, B 0.000, C 0.000 }
gfCNCPoint2[29870] = {X 81.4951, Y 12.9779, Z -3.8333, A 0.000, B 0.000, C 0.000 }
gfCNCPoint2[29871] = {X 81.4951, Y 12.1868, Z -3.8333, A 0.000, B 0.000, C 0.000 }
gfCNCPoint2[29872] = {X 81.5776, Y 11.3388, Z -3.8333, A 0.000, B 0.000, C 0.000 }
gfCNCPoint2[29873] = {X 81.8219, Y 10.5226, Z -3.8333, A 0.000, B 0.000, C 0.000 }
gfCNCPoint2[29874] = {X 82.2190, Y 9.7688, Z -3.8333, A 0.000, B 0.000, C 0.000 }
gfCNCPoint2[29875] = {X 81.8180, Y 9.5050, Z -3.8333, A 0.000, B 0.000, C 0.000 }
gfCNCPoint2[29876] = {X 68.9232, Y 9.5050, Z -3.8333, A 0.000, B 0.000, C 0.000 }
gfCNCPoint2[29877] = {X 69.1905, Y 10.7209, Z -3.8333, A 0.000, B 0.000, C 0.000 }
gfCNCPoint2[29878] = {X 69.2995, Y 11.9610, Z -3.8333, A 0.000, B 0.000, C 0.000 }
gfCNCPoint2[29879] = {X 69.3015, Y 12.0739, Z -3.8333, A 0.000, B 0.000, C 0.000 }
gfCNCPoint2[29880] = {X 69.3021, Y 12.1868, Z -3.8333, A 0.000, B 0.000, C 0.000 }
gfCNCPoint2[29881] = {X 69.3017, Y 13.0686, Z -3.8333, A 0.000, B 0.000, C 0.000 }
gfCNCPoint2[29882] = {X 69.2127, Y 14.2909, Z -3.8333, A 0.000, B 0.000, C 0.000 }
gfCNCPoint2[29883] = {X 68.9700, Y 15.4921, Z -3.8333, A 0.000, B 0.000, C 0.000 }
gfCNCPoint2[29884] = {X 73.2468, Y 26.9328, Z -3.8333, A 0.000, B 0.000, C 0.000 }
gfCNCPoint2[29885] = {X 77.7429, Y 25.2520, Z -3.8333, A 0.000, B 0.000, C 0.000 }
gfCNCPoint2[29886] = {X 77.7428, Y 18.1975, Z -3.8333, A 0.000, B 0.000, C 0.000 }
gfCNCPoint2[29887] = {X 77.0782, Y 16.9737, Z -3.8333, A 0.000, B 0.000, C 0.000 }
gfCNCPoint2[29888] = {X 76.5961, Y 15.6672, Z -3.8333, A 0.000, B 0.000, C 0.000 }
gfCNCPoint2[29889] = {X 76.3065, Y 14.3050, Z -3.8333, A 0.000, B 0.000, C 0.000 }
gfCNCPoint2[29890] = {X 74.0412, Y 14.3050, Z -3.8333, A 0.000, B 0.000, C 0.000 }
gfCNCPoint2[29891] = {X 73.9992, Y 14.7012, Z -3.8333, A 0.000, B 0.000, C 0.000 }
gfCNCPoint2[29892] = {X 73.9464, Y 15.0961, Z -3.8333, A 0.000, B 0.000, C 0.000 }
gfCNCPoint2[29893] = {X 77.7429, Y 25.2520, Z -3.8333, A 0.000, B 0.000, C 0.000 }
gfCNCPoint2[29894] = {X 75.4949, Y 26.0924, Z -3.8333, A 0.000, B 0.000, C 0.000 }
gfCNCPoint2[29895] = {X 78.9548, Y 35.3478, Z -3.8333, A 0.000, B 0.000, C 0.000 }
gfCNCPoint2[29896] = {X 79.5718, Y 35.9624, Z -3.8333, A 0.000, B 0.000, C 0.000 }
gfCNCPoint2[29897] = {X 80.1430, Y 36.6198, Z -3.8333, A 0.000, B 0.000, C 0.000 }
gfCNCPoint2[29898] = {X 80.1428, Y 17.4401, Z -3.8333, A 0.000, B 0.000, C 0.000 }
gfCNCPoint2[29899] = {X 79.4944, Y 16.4465, Z -3.8333, A 0.000, B 0.000, C 0.000 }
gfCNCPoint2[29900] = {X 79.0161, Y 15.3608, Z -3.8333, A 0.000, B 0.000, C 0.000 }
gfCNCPoint2[29901] = {X 78.7204, Y 14.2118, Z -3.8333, A 0.000, B 0.000, C 0.000 }
gfCNCPoint2[29902] = {X 78.6153, Y 13.0301, Z -3.8333, A 0.000, B 0.000, C 0.000 }
gfCNCPoint2[29903] = {X 78.6151, Y 12.1868, Z -3.8333, A 0.000, B 0.000, C 0.000 }
gfCNCPoint2[29904] = {X 78.6164, Y 12.0459, Z -3.8333, A 0.000, B 0.000, C 0.000 }
gfCNCPoint2[29905] = {X 78.6205, Y 11.9050, Z -3.8333, A 0.000, B 0.000, C 0.000 }
gfCNCPoint2[29906] = {X 71.6988, Y 11.9050, Z -3.8333, A 0.000, B 0.000, C 0.000 }
gfCNCPoint2[29907] = {X 71.7013, Y 12.0459, Z -3.8333, A 0.000, B 0.000, C 0.000 }
gfCNCPoint2[29908] = {X 71.7021, Y 12.1868, Z -3.8333, A 0.000, B 0.000, C 0.000 }
gfCNCPoint2[29909] = {X 71.7016, Y 13.0911, Z -3.8333, A 0.000, B 0.000, C 0.000 }
gfCNCPoint2[29910] = {X 71.6386, Y 14.2154, Z -3.8333, A 0.000, B 0.000, C 0.000 }
gfCNCPoint2[29911] = {X 71.4712, Y 15.3289, Z -3.8333, A 0.000, B 0.000, C 0.000 }
gfCNCPoint2[29912] = {X 75.4949, Y 26.0924, Z -3.8333, A 0.000, B 0.000, C 0.000 }
gfCNCPoint2[29913] = {X 73.2468, Y 26.9328, Z -3.8333, A 0.000, B 0.000, C 0.000 }
gfCNCPoint2[29914] = {X 76.9177, Y 36.7527, Z -3.8333, A 0.000, B 0.000, C 0.000 }
gfCNCPoint2[29915] = {X 77.6312, Y 37.4062, Z -3.8333, A 0.000, B 0.000, C 0.000 }
gfCNCPoint2[29916] = {X 78.2758, Y 38.1275, Z -3.8333, A 0.000, B 0.000, C 0.000 }
gfCNCPoint2[29917] = {X 79.0232, Y 39.1924, Z -3.8333, A 0.000, B 0.000, C 0.000 }
gfCNCPoint2[29918] = {X 79.6211, Y 40.3478, Z -3.8333, A 0.000, B 0.000, C 0.000 }
gfCNCPoint2[29919] = {X 80.0587, Y 41.5730, Z -3.8333, A 0.000, B 0.000, C 0.000 }
gfCNCPoint2[29920] = {X 80.3280, Y 42.8458, Z -3.8333, A 0.000, B 0.000, C 0.000 }
gfCNCPoint2[29921] = {X 80.4242, Y 44.1432, Z -3.8333, A 0.000, B 0.000, C 0.000 }
gfCNCPoint2[29922] = {X 80.4245, Y 45.0000, Z -3.8333, A 0.000, B 0.000, C 0.000 }
gfCNCPoint2[29923] = {X 80.3511, Y 46.1898, Z -3.8333, A 0.000, B 0.000, C 0.000 }
gfCNCPoint2[29924] = {X 80.1320, Y 47.3615, Z -3.8333, A 0.000, B 0.000, C 0.000 }
gfCNCPoint2[29925] = {X 79.7706, Y 48.4974, Z -3.8333, A 0.000, B 0.000, C 0.000 }
gfCNCPoint2[29926] = {X 79.2722, Y 49.5803, Z -3.8333, A 0.000, B 0.000, C 0.000 }
gfCNCPoint2[29927] = {X 78.4688, Y 50.8341, Z -3.8333, A 0.000, B 0.000, C 0.000 }
gfCNCPoint2[29928] = {X 77.4826, Y 51.9498, Z -3.8333, A 0.000, B 0.000, C 0.000 }
gfCNCPoint2[29929] = {X 76.3369, Y 52.9011, Z -3.8333, A 0.000, B 0.000, C 0.000 }
gfCNCPoint2[29930] = {X 75.0589, Y 53.6653, Z -3.8333, A 0.000, B 0.000, C 0.000 }
gfCNCPoint2[29931] = {X 73.6787, Y 54.2246, Z -3.8333, A 0.000, B 0.000, C 0.000 }
gfCNCPoint2[29932] = {X 72.2292, Y 54.5655, Z -3.8333, A 0.000, B 0.000, C 0.000 }
gfCNCPoint2[29933] = {X 70.7445, Y 54.6800, Z -3.8333, A 0.000, B 0.000, C 0.000 }
gfCNCPoint2[29934] = {X 64.1851, Y 54.6800, Z -3.8333, A 0.000, B 0.000, C 0.000 }
gfCNCPoint2[29935] = {X 62.7229, Y 54.5689, Z -3.8333, A 0.000, B 0.000, C 0.000 }
gfCNCPoint2[29936] = {X 61.2943, Y 54.2383, Z -3.8333, A 0.000, B 0.000, C 0.000 }
gfCNCPoint2[29937] = {X 59.9320, Y 53.6956, Z -3.8333, A 0.000, B 0.000, C 0.000 }
gfCNCPoint2[29938] = {X 58.6673, Y 52.9534, Z -3.8333, A 0.000, B 0.000, C 0.000 }
gfCNCPoint2[29939] = {X 57.5293, Y 52.0286, Z -3.8333, A 0.000, B 0.000, C 0.000 }
gfCNCPoint2[29940] = {X 56.6337, Y 51.0563, Z -3.8333, A 0.000, B 0.000, C 0.000 }
gfCNCPoint2[29941] = {X 55.8790, Y 49.9710, Z -3.8333, A 0.000, B 0.000, C 0.000 }
gfCNCPoint2[29942] = {X 55.1243, Y 51.0563, Z -3.8333, A 0.000, B 0.000, C 0.000 }
gfCNCPoint2[29943] = {X 54.2288, Y 52.0286, Z -3.8333, A 0.000, B 0.000, C 0.000 }
gfCNCPoint2[29944] = {X 53.0907, Y 52.9534, Z -3.8333, A 0.000, B 0.000, C 0.000 }
gfCNCPoint2[29945] = {X 51.8261, Y 53.6956, Z -3.8333, A 0.000, B 0.000, C 0.000 }
gfCNCPoint2[29946] = {X 50.4638, Y 54.2383, Z -3.8333, A 0.000, B 0.000, C 0.000 }
gfCNCPoint2[29947] = {X 49.0351, Y 54.5689, Z -3.8333, A 0.000, B 0.000, C 0.000 }
gfCNCPoint2[29948] = {X 47.5729, Y 54.6800, Z -3.8333, A 0.000, B 0.000, C 0.000 }
gfCNCPoint2[29949] = {X 40.6393, Y 54.6800, Z -3.8333, A 0.000, B 0.000, C 0.000 }
gfCNCPoint2[29950] = {X 39.2448, Y 54.5790, Z -3.8333, A 0.000, B 0.000, C 0.000 }
gfCNCPoint2[29951] = {X 37.8793, Y 54.2782, Z -3.8333, A 0.000, B 0.000, C 0.000 }
gfCNCPoint2[29952] = {X 36.5715, Y 53.7838, Z -3.8333, A 0.000, B 0.000, C 0.000 }
gfCNCPoint2[29953] = {X 35.3485, Y 53.1062, Z -3.8333, A 0.000, B 0.000, C 0.000 }
gfCNCPoint2[29954] = {X 33.9153, Y 54.1343, Z -3.8333, A 0.000, B 0.000, C 0.000 }
gfCNCPoint2[29955] = {X 32.3644, Y 54.9742, Z -3.8333, A 0.000, B 0.000, C 0.000 }
gfCNCPoint2[29956] = {X 30.7202, Y 55.6128, Z -3.8333, A 0.000, B 0.000, C 0.000 }
gfCNCPoint2[29957] = {X 29.0089, Y 56.0397, Z -3.8333, A 0.000, B 0.000, C 0.000 }
gfCNCPoint2[29958] = {X 27.2575, Y 56.2483, Z -3.8333, A 0.000, B 0.000, C 0.000 }
gfCNCPoint2[29959] = {X 24.9826, Y 57.2322, Z -3.8333, A 0.000, B 0.000, C 0.000 }
gfCNCPoint2[29960] = {X 22.6493, Y 58.0685, Z -3.8333, A 0.000, B 0.000, C 0.000 }
